	43:
		//Validate the CA group track length
		IF _XtsSystem.Environment.P_CaGroupOids[i] = _XtsSystem.AxesGroupRef.NcToPlc.CA.Common.GroupOID THEN
			IF _XtsSystem.Environment.Mc2CaGroup(UDINT_TO_UINT(i)).GetRailLength() <> _TrackCollection.Tracks.GetById(0).Length THEN
				LogSource.SourceName := 'InitializeXtsTask';
				LogMessage.Message	 := 'AxesGroupRef Length does not match Xts Track length!';
				LogMessage.MessageId := E_XtsLogMessage.SystemInitializationAxesGroupLengthMismatch;
				LogMessage.Severity	 := 3;
				_Logger.LogMessageInstance(LogSource, LogMessage);
				Trace.LogMessage(Key	   := LogSource.SourceName,
								 Value	   := LogMessage.Message,
								 MessageId := LogMessage.MessageId,
								 Severity  := LogMessage.Severity);

				_Error	 := TRUE;
				_ErrorId := E_XtsLogMessage.SystemInitializationAxesGroupLengthMismatch;
				_State	 := 65535;
			ELSE
				_State := 50;
			END_IF
		ELSE
			i := i + 1;
			IF i > _XtsSystem.Environment.P_CaGroupCount THEN
				LogSource.SourceName := 'InitializeXtsTask';
				LogMessage.Message	 := 'No CA group found!';
				LogMessage.MessageId := E_XtsLogMessage.SystemInitializationAxesGroupNotFound;
				LogMessage.Severity	 := 3;
				_Logger.LogMessageInstance(LogSource, LogMessage);
				Trace.LogMessage(Key	   := LogSource.SourceName,
								 Value	   := LogMessage.Message,
								 MessageId := LogMessage.MessageId,
								 Severity  := LogMessage.Severity);

				_Error	 := TRUE;
				_ErrorId := E_XtsLogMessage.SystemInitializationAxesGroupLengthMismatch;
				_State	 := 65535;
			END_IF
		END_IF

	50:
		_XtsUtility.Utility := _Xpu;
		_State				:= 60;

	60:
		IF PartSetup() THEN
			_XtsSystem.ManualDiagnoser.RefreshCollections := TRUE;
			_State										  := 100;
		END_IF

	100:
		LogSource.SourceName := 'InitializeXtsTask';
		LogMessage.Message	 := 'Initialization Finished.';
		LogMessage.MessageId := E_XtsLogMessage.SystemInitializationFinished;
		LogMessage.Severity	 := 1;
		_Logger.LogMessageInstance(LogSource, LogMessage);
		_Initialized	 := TRUE;
		_Busy			 := FALSE;
		_CommandExecuted := FALSE;
		_State			 := 0;
END_CASE
END_METHOD

{attribute 'monitoring':='call'}
PROPERTY Initialized : BOOL
GET
Initialized := _Initialized;
END_GET
SET
_Initialized := Initialized;
END_SET
END_PROPERTY

METHOD PRIVATE InfoServerSetup : BOOL
VAR_INPUT
END_VAR
CASE _SubState OF
	0:
		IF _XtsEnvironment.P_InfoServerCount > 0 THEN
			_InfoServer := _XtsEnvironment.InfoServerTcIo(1); //TODO: This needs to handle > 1 Infoserver
			_SubState		:= 10;
		ELSE
			InfoServerSetup := TRUE;
		END_IF
	10:
		IF _XtsEnvironment.GetInfoServerOids(TRUE) THEN
			_XtsEnvironment.GetInfoServerOids(FALSE);
			_InfoServerOTCID := _XtsEnvironment.P_InfoServerOids[1];
			_SubState := 20;
		END_IF
	20:
		IF _InfoServer.Init(TRUE,_InfoServerOTCID) THEN
			_InfoServer.Init(FALSE,_InfoServerOTCID);
			_SubState := 0;
			InfoServerSetup := TRUE;
		END_IF
END_CASE
END_METHOD

METHOD MoverSetup : BOOL
VAR
	LogSource  : TraceSourceInfo;
	LogMessage : TraceMessageInfo;
END_VAR
LogSource.SourceName := 'InitializeXtsTask';
LogMessage.Message	 := 'Mover Initialization Started.';
LogMessage.MessageId := E_XtsLogMessage.SystemMoverInitializationFinished;
LogMessage.Severity	 := 0;
_Logger.LogMessageInstance(LogSource, LogMessage);
_XtsSystem.Movers.ResetIterator();
WHILE _XtsSystem.Movers.MoveToNext DO
	IF _XtsSystem.Movers.Current.VirtualMover THEN
		CONTINUE;
	END_IF

	_XtsSystem.Movers.Current.MoverUtility := _Xpu.MoverTcIo(UDINT_TO_UINT(_XtsSystem.Movers.CurrentItem));
	_XtsSystem.Movers.Current.RefreshMoverId(_Xpu);
END_WHILE

_XtsUtilityProperties.UtilityProperties.Mover.XtsMoverType		 := _Xpu.GetMoverType();
_XtsUtilityProperties.UtilityProperties.Mover.XtsMagnetPlateType := _Xpu.GetMagnetPlateType();
MoverSetup														 := TRUE;
END_METHOD

METHOD PartSetup : BOOL
VAR_INPUT
END_VAR

VAR
	pPart	   : POINTER TO XtsPart;
	Part	   : I_XtsPart;
	_Parent	   : I_ContainModules;
	LogSource  : TraceSourceInfo;
	LogMessage : TraceMessageInfo;
END_VAR
CASE _SubState OF
	0:
		LogSource.SourceName := 'InitializeXtsTask';
		LogMessage.Message	 := 'Part Initialization Started.';
		LogMessage.MessageId := E_XtsLogMessage.SystemMoverInitializationStarted;
		LogMessage.Severity	 := 0;
		_Logger.LogMessageInstance(LogSource, LogMessage);
		IF NOT _Xpu.GetPartOids() THEN
			RETURN;
		END_IF

		IF _Xpu.P_PartCount < 1 THEN
			PartSetup := TRUE;
			RETURN;
		END_IF

		FOR i := 1 TO _Xpu.P_PartCount DO
			pPart		   := __NEW(XtsPart(Name := CONCAT('Part ', UDINT_TO_STRING(i))));
			Part		   := pPart^;
			Part.XtsPartId := UDINT_TO_UINT(i);
			Part.Utility   := _Xpu.PartTcIo(UDINT_TO_UINT(i));
			__QUERYINTERFACE(_XpuId, _Parent);
			Part.RegisterWithParent(_Parent);
			_PartCollection.Parts.AddItem(Part);
		END_FOR

		LogSource.SourceName := 'InitializeXtsTask';
		LogMessage.Message	 := CONCAT(TO_STRING(_PartCollection.Parts.Count), ' Parts Initialization Finished.');
		LogMessage.MessageId := E_XtsLogMessage.SystemPartInitializationFinished;
		LogMessage.Severity	 := 0;
		_Logger.LogMessageInstance(LogSource, LogMessage);
		PartSetup := TRUE;
		_SubState := 0;
END_CASE
END_METHOD

METHOD TrackSetup : BOOL
VAR_INPUT
END_VAR
VAR
	Track : I_XtsTrack;
	LogSource  : TraceSourceInfo;
	LogMessage : TraceMessageInfo;
	AxGroup : AXES_GROUP_REF;
END_VAR
CASE _SubState OF
	0:
		IF NOT _Xpu.GetTrackOids() THEN
			RETURN;
		END_IF

		IF NOT _TrackCollection.Tracks.IsEmpty THEN
			_TrackCollection.Tracks.Clear();
		END_IF

		LogSource.SourceName := 'InitializeXtsTask';
		LogMessage.Message	 := CONCAT(TO_STRING(_TrackCollection.Tracks.Count), ' Tracks Initialization Started.');
		LogMessage.MessageId := E_XtsLogMessage.SystemTrackInitializationStarted;
		_TrackCollection.Tracks.Create(_Xpu.P_TrackCount + 1);
		Track		   := _TrackCollection.Tracks.GetById(0);
		Track.Id	   := 0;
		Track.Length   := _Xpu.TrackTcIo(1).GetLength();
		Track.Otcid	   := 0;
		Track.Offset   := _Xpu.TrackTcIo(1).GetOffset();
		Track.Polarity := _Xpu.TrackTcIo(1).GetPolarity();
		Track.Utility  := 0;
		IF _Xpu.P_TrackCount = 0 THEN
			_SubState := 10;
			RETURN;
		END_IF

		FOR i := 1 TO _Xpu.P_TrackCount DO
			Track		   := _TrackCollection.Tracks.GetById(i);
			Track.Id	   := i;
			Track.Length   := _Xpu.TrackTcIo(UDINT_TO_UINT(i)).GetLength();
			Track.Otcid	   := _Xpu.P_TrackOids[i];
			Track.Offset   := _Xpu.TrackTcIo(UDINT_TO_UINT(i)).GetOffset();
			Track.Polarity := _Xpu.TrackTcIo(UDINT_TO_UINT(i)).GetPolarity();
			Track.Utility  := _Xpu.TrackTcIo(UDINT_TO_UINT(i));
		END_FOR

		_SubState := 10;

	10:
		_XtsSystem.Movers.ResetIterator();
		WHILE _XtsSystem.Movers.MoveToNext DO
			_XtsSystem.Movers.Current.Tracks := _TrackCollection.Tracks;
		END_WHILE

		LogSource.SourceName := 'InitializeXtsTask';
		LogMessage.Message	 := CONCAT(TO_STRING(_TrackCollection.Tracks.Count), ' Tracks Initialization Finished.');
		LogMessage.MessageId := E_XtsLogMessage.SystemTrackInitializationFinished;
		LogMessage.Severity	 := 0;
		_Logger.LogMessageInstance(LogSource, LogMessage);
		_SubState  := 0;
		TrackSetup := TRUE;
END_CASE
END_METHOD

//FB_Init is always available implicitly AND it is used primarily FOR initialization.

//The return value is not evaluated. For a specific influence, you can also declare the

//methods explicitly and provide additional code there with the standard initialization

//code. You can evaluate the return value.
METHOD FB_Init : BOOL
VAR_INPUT
	bInitRetains	: BOOL; // TRUE: the retain variables are initialized (reset warm / reset cold)
	bInCopyCode		: BOOL; // TRUE: the instance will be copied to the copy code afterward (online change)
END_VAR
_TaskName := 'Initalize Xts';
_TaskId	  := XtsSystemTaskId.INITIALIZE;
END_METHOD

METHOD Reset
_State			 := 0;
_Error			 := FALSE;
_ErrorId		 := 0;
_Busy			 := FALSE;
_CommandExecuted := FALSE;
_SubState		 := 0;
END_METHOD

{attribute 'monitoring' := 'call'}
PROPERTY XpuId : I_XtsXpuId
GET
XpuId := _XpuId;
END_GET
SET
_XpuId := XpuId;
__QUERYINTERFACE(_XpuId, _XtsSystem);
__QUERYINTERFACE(_XpuId, _PartCollection);
__QUERYINTERFACE(_XpuId, _TrackCollection);
__QUERYINTERFACE(_XpuId, _XtsUtilityProperties);
__QUERYINTERFACE(_XpuId, _XtsUtility);
__QUERYINTERFACE(_XtsSystem.TracePublisher,_Logger);
_MoverDetectTask   := _XtsSystem.XtsTasks.GetTaskById(XtsSystemTaskId.MOVER_DETECTION);
_MoverRedetectTask := _XtsSystem.XtsTasks.GetTaskById(XtsSystemTaskId.MOVER_REDETECTION);
_MoverIDTask	   := _XtsSystem.XtsTasks.GetTaskById(XtsSystemTaskId.MOVER_IDENTIFICATION);
END_SET
END_PROPERTY

END_FUNCTION_BLOCK

// _Internal/XtsSystem/Tasks/Interfaces/I_XtsInitializeTask
INTERFACE I_XtsInitializeTask EXTENDS I_XtsTask, I_Initializable, I_Resettable

END_INTERFACE

// _Internal/XtsSystem/Tasks/DisableXtsTask
{attribute 'no_explicit_call' := 'This FB is a CLASS and must be accessed using methods or properties'}
FUNCTION_BLOCK DisableXtsTask EXTENDS XtsTaskResult IMPLEMENTS I_XtsDisableTask, I_Cyclic
VAR
	_XpuId					   : I_XtsXpuId;
	_XtsSystem				   : I_XtsSystem;
	_State					   : UDINT;
	_MoverCommander			   : I_XtsMoverCommander;
	_GroupController		   : I_XtsMoverGroupController;
	_PositionTriggerCollection : I_XtsPositionTriggerCollection;
	_StationCollection		   : I_XtsStationCollection;
	_ZoneCollection			   : I_XtsZoneCollection;
	_AxesGroup				   : REFERENCE TO AXES_GROUP_REF;

	//CA Group Parameters
	_CollisionAvoidanceGroupParameters : I_CollisionAvoidanceGroupable;
END_VAR

PROPERTY AxesGroup : REFERENCE TO AXES_GROUP_REF
GET
AxesGroup REF= _AxesGroup;
END_GET
SET
_AxesGroup REF= AxesGroup;
END_SET
END_PROPERTY

METHOD CyclicLogic
VAR
	_Check	  : BOOL;
	AxesGroup : REFERENCE TO AXES_GROUP_REF;
	LogSource  : TraceSourceInfo;
	LogMessage : TraceMessageInfo;
END_VAR
CASE _State OF
	0:
		IF _CommandExecuted THEN
			_Busy	 := TRUE;
			_Error	 := FALSE;
			_ErrorId := 0;
			_GroupController.Disable();
			_State := 10;
		END_IF

	10:
		//Disable Group
		IF _GroupController.Error THEN
			_Error := TRUE;
			_State := 255;
		ELSIF NOT _GroupController.Enabled THEN
			AxesGroup REF= _AxesGroup;
			_MoverCommander.RemoveFromGroup(_XtsSystem.Movers, AxesGroup, 1);
			_State := 20;
		END_IF

	20:
		//Remove All From Group
		IF _MoverCommander.Error THEN
			_Error := TRUE;
			_State := 255;
		ELSIF NOT _MoverCommander.Busy THEN
			_MoverCommander.Disable(_XtsSystem.Movers);
			_State := 30;
		END_IF

	30:
		//Disable all movers
		IF _MoverCommander.Error THEN
			_Error := TRUE;
			_State := 255;
		ELSIF NOT _MoverCommander.Busy THEN
			_State := 40;
		END_IF

	40:
		//Disable All Stations
		IF NOT _XtsSystem.Config.CommandStationsOnDisable THEN
			LogSource.SourceName := 'DisableXtsTask';
			LogMessage.Message	 := 'Station Disable Skipped due to configuration.';
			LogMessage.MessageId := E_XtsLogMessage.SystemDisableStationSkipped;
			LogMessage.Severity	 := 0;
			_Logger.LogMessageInstance(LogSource, LogMessage);
			_State := 50;
			RETURN;
		END_IF

		_StationCollection.ResetIterator();
		_Check := TRUE;
		WHILE _StationCollection.MoveToNext DO
			_StationCollection.Current.Disable();
			_Check := _Check AND NOT _StationCollection.Current.Enabled;
		END_WHILE

		IF _Check THEN
			_State := 50;
		END_IF

	50:
		IF NOT _XtsSystem.Config.CommandPositionTriggersOnDisable THEN
			LogSource.SourceName := 'DisableXtsTask';
			LogMessage.Message	 := 'PositionTrigger Disable Skipped due to configuration.';
			LogMessage.MessageId := E_XtsLogMessage.SystemDisableStationSkipped;
			LogMessage.Severity	 := 0;
			_Logger.LogMessageInstance(LogSource, LogMessage);
			_State := 60;
			RETURN;
		END_IF

		//Disable All Position Triggers
		_PositionTriggerCollection.ResetIterator();
		_Check := TRUE;
		WHILE _PositionTriggerCollection.MoveToNext DO
			_PositionTriggerCollection.Current.Disable();
			_Check := _Check AND NOT _PositionTriggerCollection.Current.Enabled;
		END_WHILE

		IF _Check THEN
			_State := 60;
		END_IF

	60:
		_State			 := 0;
		_CommandExecuted := FALSE;
		_Busy			 := FALSE;
END_CASE
END_METHOD

METHOD Execute : I_XtsTaskResult
_CommandExecuted := TRUE;
Execute := THIS^;
END_METHOD

//FB_Init is always available implicitly and it is used primarily for initialization.

//The return value is not evaluated. For a specific influence, you can also declare the

//methods explicitly and provide additional code there with the standard initialization

//code. You can evaluate the return value.
METHOD FB_Init : BOOL
VAR_INPUT
	bInitRetains		  : BOOL; // TRUE: the retain variables are initialized (reset warm / reset cold)
	bInCopyCode			  : BOOL; // TRUE: the instance will be copied to the copy code afterward (online change)
END_VAR
_TaskName := 'Disable Xts';
_TaskId	  := XtsSystemTaskId.DISABLE;
END_METHOD

METHOD Reset
_State			 := 0;
_Error			 := FALSE;
_ErrorId		 := 0;
_Busy			 := FALSE;
_CommandExecuted := FALSE;
END_METHOD

{attribute 'monitoring' := 'call'}
PROPERTY XpuId : I_XtsXpuId
GET
XpuId := _XpuId;
END_GET
SET
_XpuId := XpuId;
__QUERYINTERFACE(_XpuId, _XtsSystem);
__QUERYINTERFACE(_XtsSystem.Parameters, _CollisionAvoidanceGroupParameters);
__QUERYINTERFACE(_XtsSystem.TracePublisher,_Logger);
_StationCollection		   := _XtsSystem.Stations;
_PositionTriggerCollection := _XtsSystem.PositionTriggers;
_ZoneCollection			   := _XtsSystem.Zones;
END_SET
END_PROPERTY

PROPERTY XtsMoverCommander : I_XtsMoverCommander
SET
_MoverCommander := XtsMoverCommander;
END_SET
END_PROPERTY

PROPERTY XtsMoverGroupController : I_XtsMoverGroupController
SET
_GroupController := XtsMoverGroupController;
END_SET
END_PROPERTY

END_FUNCTION_BLOCK

// _Internal/XtsSystem/Tasks/Interfaces/I_XtsDisableTask
INTERFACE I_XtsDisableTask EXTENDS I_XtsTask, I_ContainXtsMoverCommander, I_ContainXtsMoverGroupController, I_XtsExecutableTask, I_Resettable

PROPERTY AxesGroup : REFERENCE TO AXES_GROUP_REF
GET
END_GET
SET
END_SET
END_PROPERTY

END_INTERFACE

// _Internal/XtsSystem/Tasks/MoverDetectionTask
{attribute 'no_explicit_call' := 'This FB is a CLASS and must be accessed using methods or properties'}
FUNCTION_BLOCK MoverDetectionTask EXTENDS XtsTaskResult IMPLEMENTS I_XtsMoverDetectionTask
VAR
	_XpuId : I_XtsXpuId;
	_Xpu   : I_ContainXtsUtility;
END_VAR

METHOD Execute : I_XtsTaskResult
Execute := THIS^;
_Xpu.Utility.TriggerDetection();
END_METHOD

//FB_Init is always available implicitly and it is used primarily for initialization.

//The return value is not evaluated. For a specific influence, you can also declare the

//methods explicitly and provide additional code there with the standard initialization

//code. You can evaluate the return value.
METHOD FB_Init : BOOL
VAR_INPUT
	bInitRetains		  : BOOL; // TRUE: the retain variables are initialized (reset warm / reset cold)
	bInCopyCode			  : BOOL; // TRUE: the instance will be copied to the copy code afterward (online change)
END_VAR
_TaskName := 'Mover Detection';
_TaskId	  := XtsSystemTaskId.MOVER_DETECTION;
END_METHOD

{attribute 'monitoring' := 'call'}
PROPERTY XpuId : I_XtsXpuId
GET
XpuId := _XpuId;
END_GET
SET
VAR
	_XtsSystem	   : I_XtsSystem;
END_VAR
_XpuId := XpuId;
__QUERYINTERFACE(_XpuId, _XtsSystem);
__QUERYINTERFACE(_XtsSystem.TracePublisher, _Logger);
__QUERYINTERFACE(_XpuId, _Xpu);
END_SET
END_PROPERTY

END_FUNCTION_BLOCK

// _Internal/XtsSystem/Tasks/Interfaces/I_XtsMoverDetectionTask
INTERFACE I_XtsMoverDetectionTask EXTENDS I_XtsTask, I_XtsExecutableTask

END_INTERFACE

// _Internal/XtsSystem/Tasks/MoverRedetectionTask
{attribute 'no_explicit_call' := 'This FB is a CLASS and must be accessed using methods or properties'}
FUNCTION_BLOCK MoverRedetectionTask EXTENDS XtsTaskResult IMPLEMENTS I_XtsMoverRedetectionTask
VAR
	_XpuId : I_XtsXpuId;
	_Xpu   : I_ContainXtsUtility;
END_VAR

METHOD Execute : I_XtsTaskResult
Execute := THIS^;
_Xpu.Utility.TriggerRedetection();
END_METHOD

//FB_Init is always available implicitly and it is used primarily for initialization.

//The return value is not evaluated. For a specific influence, you can also declare the

//methods explicitly and provide additional code there with the standard initialization

//code. You can evaluate the return value.
METHOD FB_Init : BOOL
VAR_INPUT
	bInitRetains		  : BOOL; // TRUE: the retain variables are initialized (reset warm / reset cold)
	bInCopyCode			  : BOOL; // TRUE: the instance will be copied to the copy code afterward (online change)
END_VAR
_TaskName := 'Mover Redetection';
_TaskId	  := XtsSystemTaskId.MOVER_REDETECTION;
END_METHOD

{attribute 'monitoring' := 'call'}
PROPERTY XpuId : I_XtsXpuId
GET
XpuId := _XpuId;
END_GET
SET
VAR
	_XtsSystem : I_XtsSystem;
END_VAR
_XpuId := XpuId;
__QUERYINTERFACE(_XpuId, _XtsSystem);
__QUERYINTERFACE(_XtsSystem.TracePublisher, _Logger);
__QUERYINTERFACE(_XpuId, _Xpu);
END_SET
END_PROPERTY

END_FUNCTION_BLOCK

// _Internal/XtsSystem/Tasks/Interfaces/I_XtsMoverRedetectionTask
INTERFACE I_XtsMoverRedetectionTask EXTENDS I_XtsTask, I_XtsExecutableTask

END_INTERFACE

// _Internal/XtsSystem/Tasks/MoverIdentificationTask
{attribute 'no_explicit_call' := 'This FB is a CLASS and must be accessed using methods or properties'}
FUNCTION_BLOCK MoverIdentificationTask EXTENDS XtsTaskResult IMPLEMENTS I_XtsMoverIdentificationTask
VAR
	_XtsSystem : I_XtsSystem;
	_XpuId	   : I_XtsXpuId;
	_Xpu	   : I_ContainXtsUtility;
	_Movers	   : I_XtsMoverEnumerator;
END_VAR

METHOD CyclicLogic
VAR
	DetectionValid : BOOL;
END_VAR
IF _Xpu.Utility = 0 AND _XtsSystem.Initialized THEN
	//TODO: Create an event/alarm
	_Error := TRUE;
	RETURN;
END_IF

IF _Busy THEN
	_Error := _Xpu.Utility.GetHasMoverIdDetectionError();

	//TODO: Create an event/alarm
	DetectionValid := _Xpu.Utility.GetIsMoverIdDetectionValid();
	IF DetectionValid THEN
		_Movers.ResetIterator();
		WHILE _Movers.MoveToNext DO
			_Movers.Current.RefreshMoverId(_XtsSystem.Utility);
		END_WHILE
	END_IF

	_Busy := NOT (DetectionValid OR _Error);
END_IF
END_METHOD

METHOD Execute : I_XtsTaskResult
Execute := THIS^;
IF _Xpu.Utility = 0 THEN
	_Error := TRUE;

	//TODO: Trigger error/log message that Xpu Utility is 0
END_IF

//Protect against repeated calls
IF _Busy THEN
	RETURN;
END_IF

IF _Xpu.Utility.GetMoverIdDetectionMode() = MoverIdDetectionMode.Standard THEN
	_Busy := FALSE;
	_Movers.ResetIterator();
	WHILE _Movers.MoveToNext DO
		_Movers.Current.RefreshMoverId(_XtsSystem.Utility);
	END_WHILE

	RETURN;
END_IF

_Error	 := FALSE;
_ErrorId := 0;
_Busy	 := TRUE;
_Xpu.Utility.TriggerMoverIdDetection();
END_METHOD

//FB_Init is always available implicitly and it is used primarily for initialization.

//The return value is not evaluated. For a specific influence, you can also declare the

//methods explicitly and provide additional code there with the standard initialization

//code. You can evaluate the return value.
METHOD FB_Init : BOOL
VAR_INPUT
	bInitRetains		  : BOOL; // TRUE: the retain variables are initialized (reset warm / reset cold)
	bInCopyCode			  : BOOL; // TRUE: the instance will be copied to the copy code afterward (online change)
END_VAR
_TaskName := 'Mover 1 Detection';
_TaskId	  := XtsSystemTaskId.MOVER_IDENTIFICATION;
END_METHOD

{attribute 'monitoring' := 'call'}
PROPERTY XpuId : I_XtsXpuId
GET
XpuId := _XpuId;
END_GET
SET
_XpuId := XpuId;
__QUERYINTERFACE(_XpuId, _XtsSystem);
__QUERYINTERFACE(_XtsSystem.TracePublisher, _Logger);
__QUERYINTERFACE(_XtsSystem.Movers, _Movers);
__QUERYINTERFACE(_XpuId, _Xpu);
END_SET
END_PROPERTY

END_FUNCTION_BLOCK

// _Internal/XtsSystem/Properties/XtsSystemConfiguration
FUNCTION_BLOCK XtsSystemConfiguration IMPLEMENTS I_XtsSystemConfiguration
VAR
	_CommandStationsOnEnable		  : BOOL := TRUE;
	_CommandPositionTriggersOnEnable  : BOOL := TRUE;
	_CommandStationsOnDisable		  : BOOL := TRUE;
	_CommandPositionTriggersOnDisable : BOOL := TRUE;
END_VAR

{attribute 'monitoring' := 'call'}
PROPERTY CommandPositionTriggersOnDisable : BOOL
GET
CommandPositionTriggersOnDisable  := _CommandPositionTriggersOnDisable;
END_GET
SET
_CommandPositionTriggersOnDisable  := CommandPositionTriggersOnDisable;
END_SET
END_PROPERTY

{attribute 'monitoring' := 'call'}
PROPERTY CommandPositionTriggersOnEnable : BOOL
GET
CommandPositionTriggersOnEnable  := _CommandPositionTriggersOnEnable;
END_GET
SET
_CommandPositionTriggersOnEnable  := CommandPositionTriggersOnEnable;
END_SET
END_PROPERTY

{attribute 'monitoring' := 'call'}
PROPERTY CommandStationsOnDisable : BOOL
GET
CommandStationsOnDisable := _CommandStationsOnDisable;
END_GET
SET
_CommandStationsOnDisable := CommandStationsOnDisable;
END_SET
END_PROPERTY

{attribute 'monitoring' := 'call'}
PROPERTY CommandStationsOnEnable : BOOL
GET
CommandStationsOnEnable := _CommandStationsOnEnable;
END_GET
SET
_CommandStationsOnEnable := CommandStationsOnEnable;
END_SET
END_PROPERTY

END_FUNCTION_BLOCK

// _Internal/GroupController/XtsGroupController
FUNCTION_BLOCK XtsGroupController EXTENDS CyclicComponent IMPLEMENTS I_XtsMoverGroupController
VAR
	_AxesGroup	  : REFERENCE TO AXES_GROUP_REF;
	_Enabled	  : BOOL;
	_EnableGroup  : MC_GroupEnable;
	_DisableGroup : MC_GroupDisable;
	_ResetGroup	  : MC_GroupReset;
	_Status		  : MC_GroupReadStatus;
	_ErrorRead	  : MC_GroupReadError;
END_VAR

METHOD Disable
VAR_INPUT
END_VAR
_DisableGroup.Execute := TRUE;
END_METHOD

METHOD Enable
VAR_INPUT
END_VAR
_EnableGroup.Execute := TRUE;
END_METHOD

METHOD Reset
VAR_INPUT
END_VAR
_DisableGroup.Execute := FALSE;
_EnableGroup.Execute  := FALSE;
_ErrorRead.Enable	  := FALSE;
_ResetGroup.Execute	  := _Status.Error OR _Status.GroupErrorStop AND NOT _ResetGroup.Error;
END_METHOD

METHOD Accept
VAR_INPUT
	ComponentVisitor	: Core.I_ComponentVisitor;
END_VAR
ComponentVisitor.VisitComponent(THIS^);
END_METHOD

{attribute 'monitoring' := 'call'}
PROPERTY AxesGroup : REFERENCE TO AXES_GROUP_REF
GET
AxesGroup REF= _AxesGroup;
END_GET
SET
_AxesGroup REF= AxesGroup;
END_SET
END_PROPERTY

{attribute 'monitoring':='call'}
PROPERTY Busy : BOOL
GET
END_GET
END_PROPERTY

METHOD CyclicLogic
IF NOT __ISVALIDREF(_AxesGroup) THEN
	RETURN;
END_IF

_Status.Enable	  := TRUE;
_ErrorRead.Enable := _Status.Error OR _Status.GroupErrorStop AND NOT _ErrorRead.Error;
_EnableGroup(AxesGroup := _AxesGroup);
_DisableGroup(AxesGroup := _AxesGroup);
_ResetGroup(AxesGroup := _AxesGroup);
_Status(AxesGroup := _AxesGroup);
_ErrorRead(AxesGroup := _AxesGroup);
IF _ResetGroup.Done OR _ResetGroup.Error THEN
	_ResetGroup.Execute := FALSE;
END_IF

IF _DisableGroup.Done THEN
	_Enabled			  := FALSE;
	_DisableGroup.Execute := FALSE;
END_IF

IF _EnableGroup.Done THEN
	_Enabled			 := TRUE;
	_EnableGroup.Execute := FALSE;
END_IF
END_METHOD

METHOD DeregisterWithParent
VAR_INPUT
	Parent	: Core.I_ContainComponents;
END_VAR
Parent.DeregisterCyclic(THIS^);
Parent.DeregisterComponent(THIS^);
END_METHOD

{attribute 'monitoring':='call'}
PROPERTY Done : BOOL
GET
VAR
	_Done  : BOOL;
	Status : I_XtsMoverTaskResult;
END_VAR
END_GET
END_PROPERTY

{attribute 'monitoring' := 'call'}
PROPERTY Enabled : BOOL
GET
Enabled := _Enabled;
END_GET
END_PROPERTY

{attribute 'monitoring':='call'}
PROPERTY Error : BOOL
GET
Error := _Status.GroupErrorStop OR _ResetGroup.Error;
END_GET
END_PROPERTY

{attribute 'monitoring':='call'}
PROPERTY ErrorId : UDINT
GET
IF _ResetGroup.Error THEN
	ErrorId := _ResetGroup.ErrorId;
END_IF

IF _ErrorRead.Valid AND _ErrorRead.GroupErrorId <> 0 THEN
	ErrorId := _ErrorRead.GroupErrorId;
END_IF
END_GET
END_PROPERTY

{attribute 'monitoring':='call'}
PROPERTY GroupStatus : E_MoverGroupState
GET
GroupStatus := E_MoverGroupState.Disabled;
IF NOT _Status.Valid THEN
	RETURN;
END_IF

IF _Status.GroupDisabled THEN
	GroupStatus := E_MoverGroupState.Disabled;
ELSIF _Status.GroupNotReady THEN
	GroupStatus := E_MoverGroupState.NotReady;
ELSIF _Status.GroupStandby THEN
	GroupStatus := E_MoverGroupState.Standby;
ELSIF _Status.GroupMoving THEN
	GroupStatus := E_MoverGroupState.Moving;
ELSIF _Status.GroupStopping THEN
	GroupStatus := E_MoverGroupState.Stopping;
ELSIF _Status.GroupErrorStop THEN
	GroupStatus := E_MoverGroupState.Error;
END_IF
END_GET
END_PROPERTY

METHOD RegisterWithParent
VAR_INPUT
	Parent	: Core.I_ContainComponents;
END_VAR
Parent.RegisterCyclic(THIS^);
Parent.RegisterComponent(THIS^);
END_METHOD

{attribute 'monitoring' := 'call'}
PROPERTY TaskName : STRING
GET
TaskName := _Name;
END_GET
END_PROPERTY

END_FUNCTION_BLOCK

// _Internal/Collections/Parts/PartCollection/XtsPartCollection
{attribute 'no_explicit_call' := 'This FB is a CLASS and must be accessed using methods or properties'}
FUNCTION_BLOCK XtsPartCollection IMPLEMENTS I_XtsPartCollection, I_Peekable
VAR
	_Collection : Collection;
END_VAR

{attribute 'monitoring':='call'}
PROPERTY Current : I_XtsPart
GET
__QUERYINTERFACE(_Collection.Current,Current);
END_GET
END_PROPERTY

{attribute 'monitoring' := 'call'}
PROPERTY CurrentItem : UDINT
GET
CurrentItem := _Collection.CurrentItem;
END_GET
END_PROPERTY

PROPERTY MoveToNext : BOOL
GET
MoveToNext := _Collection.MoveToNext;
END_GET
END_PROPERTY

METHOD ResetIterator
_Collection.ResetIterator();
END_METHOD

METHOD AcceptPeeker
VAR_INPUT
	Peeker	: Core.I_Peeker;
END_VAR
Peeker.PeekCollection(_Collection);
END_METHOD

METHOD AddItem
VAR_INPUT
	Part : I_XtsPart;
END_VAR
_Collection.AddItem(Part);
END_METHOD

METHOD Clear
VAR_INPUT
END_VAR
_Collection.Clear();
END_METHOD

{attribute 'monitoring' := 'call'}
PROPERTY Count : UDINT
GET
Count := _Collection.Count;
END_GET
END_PROPERTY

//FB_Exit must be implemented explicitly. If there is an implementation, then the
//method is called before the controller removes the code of the function block instance
//(implicit call). The return value is not evaluated.
METHOD FB_Exit: BOOL
VAR_INPUT
    bInCopyCode: BOOL;  // TRUE: the exit method is called in order to leave the instance which will be copied afterwards (online change).  
END_VAR
IF bInCopyCode OR IsEmpty THEN
	RETURN;
END_IF

ResetIterator();
WHILE MoveToNext DO
	Current.Dispose();
END_WHILE
Clear();
END_METHOD

METHOD GetById : I_XtsPart
VAR_INPUT
	PartId : UDINT;
END_VAR
VAR
	_Part : I_XtsPart;
END_VAR
GetById := NullObjects.XtsPart;
_Collection.ResetIterator();
WHILE _Collection.MoveToNext DO
	__QUERYINTERFACE(_Collection.Current,_Part);
	IF _Part.XtsPartId = UDINT_TO_UINT(PartId) THEN
		GetById := _Part;
		RETURN;
	END_IF
END_WHILE
END_METHOD

METHOD GetByOtcid : I_XtsPart
VAR_INPUT
	PartOtcid : OTCID;
END_VAR
VAR
	_Part : I_XtsPart;
END_VAR
__QUERYINTERFACE(NullObjects.XtsPart, GetByOtcid);
_Collection.ResetIterator();
WHILE _Collection.MoveToNext DO
	__QUERYINTERFACE(_Collection.Current, _Part);
	IF _Part.Properties.General.OTCID = PartOtcid THEN
		GetByOtcid := _Part;
		RETURN;
	END_IF
END_WHILE
END_METHOD

{attribute 'monitoring':='call'}
PROPERTY IsEmpty : BOOL
GET
IsEmpty := _Collection.IsEmpty;
END_GET
END_PROPERTY

METHOD Remove
VAR_INPUT
	Part : I_XtsPart;
END_VAR
_Collection.RemoveItem(Part);
END_METHOD

END_FUNCTION_BLOCK

// _Internal/XtsSystem/Status/XtsSystemStatus
{attribute 'no_explicit_call' := 'This FB is a CLASS and must be accessed using methods or properties'}
FUNCTION_BLOCK XtsSystemStatus IMPLEMENTS I_XtsSystemStatus
VAR
	_XtsSystem			 : I_XtsSystem;
	_Vdc24Okay			 : BOOL;
	_Vdc48Okay			 : BOOL;
	_PartReadyCounter	 : USINT;
	_PartNotReadyCounter : USINT;
END_VAR

METHOD CyclicLogic
VAR
	Part : I_XtsPart;
END_VAR
//TODO: Split this into a seperate set of commands
_Vdc24Okay := _XtsSystem.Utility.GetIsDcLinkVoltageReady();
_Vdc48Okay := _XtsSystem.Utility.GetIsDcLinkVoltageReady();
END_METHOD

//FB_Init is always available implicitly and it is used primarily for initialization.

//The return value is not evaluated. For a specific influence, you can also declare the

//methods explicitly and provide additional code there with the standard initialization

//code. You can evaluate the return value.
METHOD FB_Init : BOOL
VAR_INPUT
	bInitRetains : BOOL; // TRUE: the retain variables are initialized (reset warm / reset cold)
	bInCopyCode	 : BOOL; // TRUE: the instance will be copied to the copy code afterward (online change)   
	XtsSystem	 : I_XtsSystem;
END_VAR
_XtsSystem := XtsSystem;
END_METHOD

{attribute 'monitoring' := 'call'}
PROPERTY NumberOfMovers : UDINT
GET
NumberOfMovers := _XtsSystem.Movers.Count;
END_GET
END_PROPERTY

{attribute 'monitoring' := 'call'}
PROPERTY NumberOfParts : UDINT
GET
NumberOfParts := _XtsSystem.Parts.Count;
END_GET
END_PROPERTY

{attribute 'monitoring' := 'call'}
PROPERTY NumberOfPositionTriggers : UDINT
GET
NumberOfPositionTriggers := _XtsSystem.PositionTriggers.Count;
END_GET
END_PROPERTY

{attribute 'monitoring' := 'call'}
PROPERTY NumberOfStations : UDINT
GET
NumberOfStations := _XtsSystem.Stations.Count;
END_GET
END_PROPERTY

{attribute 'monitoring' := 'call'}
PROPERTY NumberOfTracks : UDINT
GET
NumberOfTracks := _XtsSystem.Tracks.Count;
END_GET
END_PROPERTY

{attribute 'monitoring' := 'call'}
PROPERTY NumberOfZones : UDINT
GET
NumberOfZones := _XtsSystem.Zones.Count;
END_GET
END_PROPERTY

{attribute 'monitoring':='call'}
PROPERTY NumberPartsNotReady : USINT
GET
NumberPartsNotReady := _PartNotReadyCounter;
END_GET
END_PROPERTY

{attribute 'monitoring':='call'}
PROPERTY NumberPartsReady : USINT
GET
NumberPartsReady := _PartReadyCounter;
END_GET
END_PROPERTY

{attribute 'monitoring':='call'}
PROPERTY Simulated : BOOL
GET
IF _XtsSystem.Utility = 0 THEN
	RETURN;
END_IF

Simulated := _XtsSystem.Utility.GetOperationMode() = OperationMode.Simulation;
END_GET
END_PROPERTY

{attribute 'monitoring':='call'}
PROPERTY Vdc24Okay : BOOL
GET
VAR
	VoltageOk : BOOL;
END_VAR
Vdc24Okay := _Vdc24Okay;
END_GET
END_PROPERTY

{attribute 'monitoring':='call'}
PROPERTY Vdc48Okay : BOOL
GET
Vdc48Okay := _Vdc48Okay;
END_GET
END_PROPERTY

END_FUNCTION_BLOCK

// _Internal/Collections/Tracks/TrackCollection/XtsTrackCollection
{attribute 'no_explicit_call' := 'This FB is a CLASS and must be accessed using methods or properties'}
{attribute 'hide_all_locals}
FUNCTION_BLOCK XtsTrackCollection IMPLEMENTS I_XtsTrackCollection
VAR
	pTrackBuffer	: POINTER TO PVOID;
	_NumberOfTracks : UINT;
	_CurrentTrack : I_XtsTrack;
	_CurrentIndex : UDINT := 0;
END_VAR

METHOD Clear
VAR
	i	   : UDINT;
	Track : POINTER TO XtsTrack;
END_VAR
IF IsEmpty THEN
	RETURN;
END_IF

FOR i := 0 TO _NumberOfTracks - 1 DO
	Track := GetTrackInstance(i);
	Track^.Dispose();
END_FOR

__DELETE(pTrackBuffer);
_NumberOfTracks := 0;
END_METHOD

{attribute 'monitoring' := 'call'}
PROPERTY Count : UDINT
GET
Count := _NumberOfTracks;
END_GET
END_PROPERTY

{attribute 'hide'}
METHOD Create : BOOL
VAR_INPUT
	NumberOfTracks : UINT;
END_VAR
VAR
	i		 : UINT;
	pTrack	 : POINTER TO XtsTrack;
	ppBuffer : POINTER TO POINTER TO XtsTrack;
END_VAR
IF NOT IsEmpty THEN
	Clear();
END_IF

_NumberOfTracks := NumberOfTracks;
pTrackBuffer	:= __NEW(PVOID, _NumberOfTracks);
IF pTrackBuffer <> 0 THEN
	FOR i := 0 TO _NumberOfTracks - 1 DO
		pTrack	  := __NEW(XtsTrack);
		ppBuffer  := pTrackBuffer + (i * SIZEOF(PVOID));
		ppBuffer^ := pTrack;
	END_FOR

	Create := TRUE;
END_IF
END_METHOD

METHOD GetById : I_XtsTrack
VAR_INPUT
	TrackId : UDINT;
END_VAR
GetById := GetTrackInstance(TrackId)^;
END_METHOD

METHOD GetByOtcid : I_XtsTrack
VAR_INPUT
	TrackOtcid : OTCID;
END_VAR
VAR
	i : UDINT;
	ppTrack : POINTER TO POINTER TO XtsTrack;
END_VAR
GetByOtcid := NullObjects.XtsTrack;
FOR i := 0 TO _NumberOfTracks - 1 DO
	ppTrack := pTrackBuffer + ((i) * SIZEOF(PVOID));
	IF ppTrack^^.Otcid = TrackOtcid THEN
		GetByOtcid := ppTrack^^;
		RETURN;
	END_IF
END_FOR
END_METHOD

{attribute 'monitoring' := 'call'}
PROPERTY IsEmpty : BOOL
GET
IsEmpty := _NumberOfTracks = 0;
END_GET
END_PROPERTY

{attribute 'monitoring' := 'call'}
PROPERTY Current : I_XtsTrack
GET
IF  _CurrentTrack = 0 THEN
	Current := NullObjects.XtsTrack;
ELSE
	Current := _CurrentTrack;
END_IF
END_GET
END_PROPERTY

{attribute 'monitoring' := 'call'}
PROPERTY CurrentIndex : UDINT
GET
CurrentIndex := _CurrentIndex;
END_GET
END_PROPERTY

PROPERTY MoveToNext : BOOL
GET
MoveToNext := FALSE;
IF _NumberOfTracks = 0 THEN
	RETURN;
END_IF

IF _CurrentIndex = _NumberOfTracks THEN
	RETURN;
END_IF

_CurrentTrack := GetById(_CurrentIndex + 1);
_CurrentIndex := _CurrentIndex + 1;
MoveToNext	  := TRUE;
END_GET
END_PROPERTY

METHOD ResetIterator
_CurrentTrack := NullObjects.XtsTrack;
_CurrentIndex := 0;
END_METHOD

METHOD PROTECTED CheckTrackId : BOOL
VAR_INPUT
	TrackId : UDINT;
END_VAR
CheckTrackId := (TrackId >= 0) AND (TrackId < _NumberOfTracks) AND (pTrackBuffer <> 0);
END_METHOD

METHOD PROTECTED GetTrackInstance : POINTER TO XtsTrack
VAR_INPUT
	TrackId : UDINT;
END_VAR

VAR
	ppTrack : POINTER TO POINTER TO XtsTrack;
END_VAR
IF CheckTrackId(TrackId) THEN
	ppTrack := pTrackBuffer + ((TrackId) * SIZEOF(PVOID));
	GetTrackInstance := ppTrack^;
ELSE
	GetTrackInstance := ADR(NullObjects.XtsTrack);
END_IF
END_METHOD

//FB_Exit must be implemented explicitly. If there is an implementation, then the
//method is called before the controller removes the code of the function block instance
//(implicit call). The return value is not evaluated.
METHOD FB_Exit: BOOL
VAR_INPUT
    bInCopyCode: BOOL;  // TRUE: the exit method is called in order to leave the instance which will be copied afterwards (online change).  
END_VAR
IF bInCopyCode THEN
	RETURN;
END_IF

Clear();
END_METHOD

END_FUNCTION_BLOCK

// _Internal/XtsSystem/Properties/XtsSystemUtilityProperties
{attribute 'no_explicit_call' := 'This FB is a CLASS and must be accessed using methods or properties'}
FUNCTION_BLOCK XtsSystemUtilityProperties IMPLEMENTS I_XtsSystemUtilityProperties
VAR
	_Mover : XtsSystemUtilityPropertiesMover;
END_VAR

PROPERTY Mover : I_XtsSystemUtilityPropertiesMover
GET
Mover := _Mover;
END_GET
END_PROPERTY

END_FUNCTION_BLOCK

// _Internal/XtsSystem/Properties/XtsSystemUtilityPropertiesMover
{attribute 'no_explicit_call' := 'This FB is a CLASS and must be accessed using methods or properties'}
FUNCTION_BLOCK XtsSystemUtilityPropertiesMover IMPLEMENTS I_XtsSystemUtilityPropertiesMover
VAR
	_MagnetPlate : MagnetPlateType;
	_MoverType	 : MoverType;
END_VAR

PROPERTY XtsMagnetPlateType : MagnetPlateType
GET
XtsMagnetPlateType := _MagnetPlate;
END_GET
SET
_MagnetPlate := XtsMagnetPlateType;
END_SET
END_PROPERTY

PROPERTY XtsMoverType : MoverType
GET
XtsMoverType := _MoverType;
END_GET
SET
_MoverType := XtsMoverType;
END_SET
END_PROPERTY

END_FUNCTION_BLOCK

// _Internal/Collections/Movers/MoverList/Interfaces/I_XtsMoverList
INTERFACE I_XtsMoverList EXTENDS I_XtsMoverCollection

METHOD Contains : BOOL
VAR_INPUT
	Mover : I_XtsMover;
END_VAR
END_METHOD

METHOD GetAtIndex : I_XtsMover
VAR_INPUT
	Index : UDINT; //0 indexed
END_VAR
END_METHOD

METHOD InsertAtIndex
VAR_INPUT
	Mover : I_XtsMover;
	Index : UDINT;
END_VAR
END_METHOD

METHOD RemoveAtIndex
VAR_INPUT
	MoverIndex : UDINT;
END_VAR
END_METHOD

END_INTERFACE

// _Internal/Collections/Movers/MoverList/XtsMoverList
{attribute 'no_explicit_call' := 'This FB is a CLASS and must be accessed using methods or properties'}
FUNCTION_BLOCK XtsMoverList IMPLEMENTS I_XtsMoverList
VAR
	_List : List;
END_VAR

METHOD AcceptMoverVisitor
VAR_INPUT
	MoverVisitor : I_XtsMoverVisitor;
END_VAR
VAR
	Mover : I_XtsMover;
END_VAR
_List.ResetIterator();
WHILE _List.MoveToNext DO
	__QUERYINTERFACE(_List.Current, Mover);
	Mover.AcceptMoverVisitor(MoverVisitor);
END_WHILE
END_METHOD

METHOD AddItem
VAR_INPUT
	Mover	: I_XtsMover;
END_VAR
_List.AddItem(Mover);
END_METHOD

METHOD Clear
_List.Clear();
END_METHOD

{attribute 'monitoring' := 'call'}
PROPERTY Count : UDINT
GET
Count := _List.Count;
END_GET
END_PROPERTY

{attribute 'monitoring' := 'call'}
PROPERTY IsEmpty : BOOL
GET
IsEmpty := _List.IsEmpty;
END_GET
END_PROPERTY

METHOD Map
VAR_INPUT
	Validator : I_XtsMoverValidator;
	Visitor	  : I_XtsMoverVisitor;
END_VAR
VAR
	Mover : I_XtsMover;
END_VAR
_List.ResetIterator();
WHILE _List.MoveToNext DO
	__QUERYINTERFACE(_List.Current, Mover);
	IF Validator.Valid(Mover) THEN
		Visitor.VisitMover(Mover);
	END_IF
END_WHILE
END_METHOD

METHOD Remove
VAR_INPUT
	Mover	: I_XtsMover;
END_VAR
_List.RemoveItem(Mover);
END_METHOD

{attribute 'monitoring':='call'}
PROPERTY Current : I_XtsMover
GET
VAR
	Mover : I_XtsMover;
END_VAR
__QUERYINTERFACE(_List.Current,Mover);
Current := Mover;
END_GET
END_PROPERTY

{attribute 'monitoring' := 'call'}
PROPERTY CurrentItem : UDINT
GET
CurrentItem := _List.CurrentItem;
END_GET
END_PROPERTY

PROPERTY MoveToNext : BOOL
GET
MoveToNext := _List.MoveToNext;
END_GET
END_PROPERTY

METHOD ResetIterator
_List.ResetIterator();
END_METHOD

METHOD Contains : BOOL
VAR_INPUT
	Mover	: I_XtsMover;
END_VAR
IF _List.Count = 0 THEN
	Contains := FALSE;
	RETURN;
END_IF
Contains := _List.ContainsItem(Mover);
END_METHOD

//FB_Exit must be implemented explicitly. If there is an implementation, then the
//method is called before the controller removes the code of the function block instance
//(implicit call). The return value is not evaluated.
METHOD FB_Exit: BOOL
VAR_INPUT
    bInCopyCode: BOOL;  // TRUE: the exit method is called in order to leave the instance which will be copied afterwards (online change).  
END_VAR
_List.FB_Exit(bInCopyCode);
END_METHOD

METHOD GetAtIndex : I_XtsMover
VAR_INPUT
	Index : UDINT; //0 based
END_VAR
__QUERYINTERFACE(_List.GetAtIndex(Index), GetAtIndex);
END_METHOD

METHOD InsertAtIndex
VAR_INPUT
	Mover : I_XtsMover;
	Index : UDINT;
END_VAR
_List.InsertAtIndex(Mover, Index);
END_METHOD

{attribute 'monitoring':='call'}
PROPERTY Movers : I_XtsMoverCollection
GET
Movers := THIS^;
END_GET
END_PROPERTY

METHOD RemoveAtIndex
VAR_INPUT
	MoverIndex	: UDINT;
END_VAR
_List.RemoveAtIndex(MoverIndex);
END_METHOD

END_FUNCTION_BLOCK

// _Internal/Collections/Movers/MoverQueue/XtsMoverQueue
{attribute 'no_explicit_call' := 'This FB is a CLASS and must be accessed using methods or properties'}
FUNCTION_BLOCK XtsMoverQueue IMPLEMENTS I_XtsMoverQueue
VAR
	_Queue			 : XtsMoverList;
END_VAR

{attribute 'monitoring':='call'}
PROPERTY Current : I_XtsMover
GET
Current := _Queue.Current;
END_GET
END_PROPERTY

{attribute 'monitoring' := 'call'}
PROPERTY CurrentItem : UDINT
GET
CurrentItem := _Queue.CurrentItem;
END_GET
END_PROPERTY

METHOD Map
VAR_INPUT
	Validator : I_XtsMoverValidator;
	Visitor	  : I_XtsMoverVisitor;
END_VAR
VAR
	Mover : I_XtsMover;
END_VAR
_Queue.ResetIterator();
WHILE _Queue.MoveToNext DO
	__QUERYINTERFACE(_Queue.Current, Mover);
	IF Validator.Valid(Mover) THEN
		Visitor.VisitMover(Mover);
	END_IF
END_WHILE
END_METHOD

PROPERTY MoveToNext : BOOL
GET
MoveToNext := _Queue.MoveToNext;
END_GET
END_PROPERTY

METHOD ResetIterator
_Queue.ResetIterator();
END_METHOD

METHOD AcceptMoverVisitor
VAR_INPUT
	MoverVisitor : I_XtsMoverVisitor;
END_VAR
VAR
	Mover : I_XtsMover;
END_VAR
_Queue.ResetIterator();
WHILE _Queue.MoveToNext DO
	__QUERYINTERFACE(_Queue.Current, Mover);
	Mover.AcceptMoverVisitor(MoverVisitor);
END_WHILE
END_METHOD

METHOD Clear
_Queue.Clear();
END_METHOD

{attribute 'monitoring':='call'}
PROPERTY Count : UDINT
GET
Count := _Queue.Count;
END_GET
END_PROPERTY

METHOD Dequeue : I_XtsMover
IF Count = 0 THEN
	RETURN;
END_IF
__QUERYINTERFACE(_Queue.GetAtIndex(0),Dequeue);
_Queue.RemoveAtIndex(0);
END_METHOD

METHOD Enqueue
VAR_INPUT
	Mover	: I_XtsMover;
END_VAR
_Queue.AddItem(Mover);
END_METHOD

//FB_Exit must be implemented explicitly. If there is an implementation, then the
//method is called before the controller removes the code of the function block instance
//(implicit call). The return value is not evaluated.
METHOD FB_Exit: BOOL
VAR_INPUT
    bInCopyCode: BOOL;  // TRUE: the exit method is called in order to leave the instance which will be copied afterwards (online change).  
END_VAR
_Queue.FB_Exit(bInCopyCode);
END_METHOD

{attribute 'monitoring':='call'}
PROPERTY Movers : I_XtsMoverCollection
GET
Movers := _Queue;
END_GET
END_PROPERTY

METHOD Peek : I_XtsMover
IF Count = 0 THEN
	RETURN;
END_IF
__QUERYINTERFACE(_Queue.GetAtIndex(0),Peek);
END_METHOD

END_FUNCTION_BLOCK

// _Internal/Collections/Movers/MoverQueue/XtsMoverUniqueQueue
{attribute 'no_explicit_call' := 'This FB is a CLASS and must be accessed using methods or properties'}
FUNCTION_BLOCK XtsMoverUniqueQueue EXTENDS XtsMoverQueue
VAR
END_VAR

METHOD Enqueue
VAR_INPUT
	Mover	: I_XtsMover;
END_VAR
IF _Queue.Contains(Mover) THEN
	RETURN;
END_IF
_Queue.AddItem(Mover);
END_METHOD

END_FUNCTION_BLOCK

// _Internal/Collections/I_ContainXtsMoverList
INTERFACE I_ContainXtsMoverList EXTENDS I_Base

{attribute 'monitoring':='call'}
PROPERTY Movers : I_XtsMoverList
GET
END_GET
END_PROPERTY

END_INTERFACE

// _Internal/Collections/I_OperatesOnMovers
INTERFACE I_OperatesOnMovers EXTENDS I_Base

PROPERTY Movers : I_XtsMoverCollection
SET
END_SET
END_PROPERTY

END_INTERFACE

// _Internal/Frames/Interfaces/I_BaseFrame
INTERFACE I_BaseFrame EXTENDS I_Base

{attribute 'monitoring':='call'}
PROPERTY FrameName : STRING
GET
END_GET
SET
END_SET
END_PROPERTY

END_INTERFACE

// _Internal/Frames/Interfaces/I_FrameModulo
INTERFACE I_FrameModulo EXTENDS I_Base

{attribute 'monitoring' := 'call'}
PROPERTY ModuloLength : LREAL
GET
END_GET
SET
END_SET
END_PROPERTY

END_INTERFACE

// _Internal/Frames/Interfaces/I_FrameOffset
INTERFACE I_FrameOffset EXTENDS I_Base

{attribute 'monitoring' := 'call'}
PROPERTY OffsetToParent : LREAL
GET
END_GET
SET
END_SET
END_PROPERTY

END_INTERFACE

// _Internal/Frames/Interfaces/I_HasAReferenceFrame
INTERFACE I_HasAReferenceFrame EXTENDS I_Base

{attribute 'monitoring' := 'call'}
PROPERTY ReferenceFrame : I_ReferenceFrame
GET
END_GET
END_PROPERTY

METHOD SetReferenceFrame
VAR_INPUT
	ReferenceFrame : I_ReferenceFrame;
END_VAR
END_METHOD

END_INTERFACE

// _Internal/Frames/ReferenceFrame
{attribute 'no_explicit_call' := 'This FB is a CLASS and must be accessed using methods or properties'}
FUNCTION_BLOCK ReferenceFrame IMPLEMENTS I_ReferenceFrame
VAR
	{attribute 'hide'}
	NullReferenceFrame : NullReferenceFrame;
	_FrameName		   : T_MaxString;
	_OffsetToParent	   : LREAL;
	_ModuloLength	   : LREAL;
	_ReferenceFrame	   : I_ReferenceFrame := NullReferenceFrame;
END_VAR

//FB_Init is always available implicitly and it is used primarily for initialization.

//The return value is not evaluated. For a specific influence, you can also declare the

//methods explicitly and provide additional code there with the standard initialization

//code. You can evaluate the return value.
METHOD FB_Init : BOOL
VAR_INPUT
	bInitRetains   : BOOL; // TRUE: the retain variables are initialized (reset warm / reset cold)
	bInCopyCode	   : BOOL; // TRUE: the instance will be copied to the copy code afterward (online change)
	FrameName		   : T_MaxString;
	Offset		   : LREAL;
	ModuloLength   : LREAL;
	ReferenceFrame : I_ReferenceFrame;
END_VAR
_FrameName	  := FrameName;
_OffsetToParent		  := Offset;
_ModuloLength := ModuloLength;
IF ReferenceFrame <> 0 THEN
	_ReferenceFrame := ReferenceFrame;
END_IF
END_METHOD

{attribute 'monitoring' := 'call'}
PROPERTY FrameName : STRING
GET
FrameName := _FrameName;
END_GET
SET
FrameName := _FrameName;
END_SET
END_PROPERTY

{attribute 'monitoring' := 'call'}
PROPERTY ModuloLength : LREAL
GET
ModuloLength := _ModuloLength;
END_GET
SET
_ModuloLength := ModuloLength;
END_SET
END_PROPERTY

{attribute 'hide'}
PROPERTY OffsetToGlobal : LREAL
GET
OffsetToGlobal := _OffsetToParent + _ReferenceFrame.OffsetToGlobal;
END_GET
END_PROPERTY

{attribute 'monitoring' := 'call'}
PROPERTY OffsetToParent : LREAL
GET
OffsetToParent := _OffsetToParent;
END_GET
SET
_OffsetToParent := OffsetToParent;
END_SET
END_PROPERTY

{attribute 'monitoring' := 'call'}
PROPERTY ReferenceFrame : I_ReferenceFrame
GET
ReferenceFrame := _ReferenceFrame;
END_GET
END_PROPERTY

METHOD SetReferenceFrame 
VAR_INPUT
	ReferenceFrame	: I_ReferenceFrame;
END_VAR
_ReferenceFrame := ReferenceFrame;
END_METHOD

END_FUNCTION_BLOCK

// _Internal/Frames/Interfaces/I_ReferenceFrame
INTERFACE I_ReferenceFrame EXTENDS I_BaseFrame,I_FrameModulo,I_FrameOffset, I_HasAReferenceFrame, I_InGlobalSpace

END_INTERFACE

// _Internal/Frames/Interfaces/I_InGlobalSpace
INTERFACE I_InGlobalSpace EXTENDS I_Base

{attribute 'hide'}
PROPERTY OffsetToGlobal : LREAL
GET
END_GET
END_PROPERTY

END_INTERFACE

// _Internal/NullObjects/NullReferenceFrame
{attribute 'no_explicit_call' := 'This FB is a CLASS and must be accessed using methods or properties'}
{attribute 'conditionalshow'}
{warning disable C0094}
{warning disable C0568}
FUNCTION_BLOCK NullReferenceFrame IMPLEMENTS I_ReferenceFrame, I_NullObject
VAR
END_VAR

{attribute 'monitoring' := 'call'}
PROPERTY FrameName : STRING
GET
FrameName := 'Null Frame';
END_GET
SET
END_SET
END_PROPERTY

PROPERTY ModuloLength : LREAL
GET
END_GET
SET
END_SET
END_PROPERTY

PROPERTY OffsetToGlobal : LREAL
GET
END_GET
END_PROPERTY

PROPERTY OffsetToParent : LREAL
GET
END_GET
SET
END_SET
END_PROPERTY

PROPERTY ReferenceFrame : I_ReferenceFrame
GET
END_GET
END_PROPERTY

METHOD SetReferenceFrame
VAR_INPUT
	ReferenceFrame	: I_ReferenceFrame;
END_VAR
END_METHOD

END_FUNCTION_BLOCK

// _Internal/Frames/Interfaces/I_ReferencedPosition
INTERFACE I_ReferencedPosition EXTENDS I_Base, I_Positionable,I_HasAReferenceFrame

END_INTERFACE

// _Internal/Frames/ReferencedPosition
{attribute 'no_explicit_call' := 'This FB is a CLASS and must be accessed using methods or properties'}
FUNCTION_BLOCK ReferencedPosition IMPLEMENTS I_ReferencedPosition
VAR
	{attribute 'hide'}
	NullReferenceFrame : NullReferenceFrame;
	_GlobalPosition	   : LREAL;
	_CurrentFrame	   : I_ReferenceFrame := NullReferenceFrame;
	
	//
	_CurrentPosition   : LREAL;
END_VAR

{attribute 'monitoring' := 'call'}
PROPERTY Position : LREAL
GET
VAR
	tmp : LREAL;
END_VAR
tmp := _GlobalPosition - _CurrentFrame.OffsetToGlobal;
//If my current frame is modulo'd, return the position in that modulo
IF _CurrentFrame.ModuloLength <> 0.0 THEN
    tmp := tmp - _CurrentFrame.ModuloLength * TRUNC(tmp / _CurrentFrame.ModuloLength);
    IF tmp < 0.0 THEN
        tmp := tmp + _CurrentFrame.ModuloLength;
    END_IF; 
END_IF;
Position := tmp;
END_GET
SET
_GlobalPosition := Position + _CurrentFrame.OffsetToGlobal;
END_SET
END_PROPERTY

{attribute 'monitoring' := 'call'}
PROPERTY ReferenceFrame : I_ReferenceFrame
GET
END_GET
END_PROPERTY

METHOD SetReferenceFrame 
VAR_INPUT
	ReferenceFrame	: I_ReferenceFrame;
END_VAR
_CurrentFrame := ReferenceFrame;
END_METHOD

END_FUNCTION_BLOCK

// _Internal/NullObjects/NullAxisRef
{attribute 'no_explicit_call' := 'This FB is a CLASS and must be accessed using methods or properties'}
{attribute 'conditionalshow'}
{warning disable C0094}
FUNCTION_BLOCK NullAxisRef IMPLEMENTS I_AxisRef,I_NullObject
VAR
	NullAxis : AXIS_REF;
END_VAR

PROPERTY Axis : REFERENCE TO Tc2_MC2.AXIS_REF
GET
Axis REF= NullAxis;
END_GET
END_PROPERTY

END_FUNCTION_BLOCK

// _Internal/NullObjects/NullMechatronicsLocalLog
{attribute 'no_explicit_call' := 'This FB is a CLASS and must be accessed using methods or properties'}
{attribute 'conditionalshow'}
{warning disable C0094}
FUNCTION_BLOCK NullMechatronicsLocalLog IMPLEMENTS I_XtsLocalLog, I_NullObject
VAR
END_VAR

METHOD Clear
VAR_INPUT
END_VAR
END_METHOD

{attribute 'monitoring':='call'}
PROPERTY Commands : REFERENCE TO ARRAY[0..XtsCoreParameters.MAX_NUMBER_LOCAL_LOG - 1] OF T_MaxString
GET
END_GET
END_PROPERTY

{attribute 'monitoring':='call'}
PROPERTY DetailedCommands : REFERENCE TO ARRAY[0..XtsCoreParameters.MAX_NUMBER_LOCAL_LOG - 1] OF I_XtsLogCommand
GET
END_GET
END_PROPERTY

END_FUNCTION_BLOCK

// _Internal/NullObjects/NullMechatronicsLogger
{attribute 'no_explicit_call' := 'This FB is a CLASS and must be accessed using methods or properties'}
{attribute 'conditionalshow'}
{warning disable C0094}
FUNCTION_BLOCK NullMechatronicsLogger IMPLEMENTS I_XtsLogger, I_NullObject
VAR
END_VAR

METHOD LogMessage
VAR_INPUT
	Key	: Core.T_MaxString;
	Value	: Core.T_MaxString;
	SourceId	: UDINT := 0;
	TimeStamp	: ULINT := 0;
	MessageId	: UDINT := 1;
	Severity	: USINT := 1;
END_VAR
END_METHOD

METHOD LogMessageInstance
VAR_INPUT
	SourceInfo	: Core.I_TraceSourceInfo;
	MessageInfo	: Core.I_TraceMessageInfo;
	Arguments	: Core.I_TraceArgument := 0;
END_VAR
END_METHOD

END_FUNCTION_BLOCK

// _Internal/NullObjects/NullMechatronicsTracePublisher
{attribute 'no_explicit_call' := 'This FB is a CLASS and must be accessed using methods or properties'}
{attribute 'conditionalshow'}
{warning disable C0094}
FUNCTION_BLOCK NullMechatronicsTracePublisher IMPLEMENTS I_XtsTracePublisher, I_NullObject
VAR
END_VAR

METHOD LogMessage
VAR_INPUT
	Key	: Core.T_MaxString;
	Value	: Core.T_MaxString;
	SourceId	: UDINT := 0;
	TimeStamp	: ULINT := 0;
	MessageId	: UDINT := 1;
	Severity	: USINT := 1;
END_VAR
END_METHOD

METHOD LogMessageInstance
VAR_INPUT
	SourceInfo	: Core.I_TraceSourceInfo;
	MessageInfo	: Core.I_TraceMessageInfo;
	Arguments	: Core.I_TraceArgument := 0;
END_VAR
END_METHOD

METHOD Subscribe
VAR_INPUT
	Logger : I_XtsLogger;
END_VAR
END_METHOD

METHOD Unsubscribe
VAR_INPUT
	Logger : I_XtsLogger;
END_VAR
END_METHOD

END_FUNCTION_BLOCK

// _Internal/NullObjects/NullMoverCollection
{attribute 'no_explicit_call' := 'This FB is a CLASS and must be accessed using methods or properties'}
{attribute 'conditionalshow'}
{warning disable C0094}
{warning disable C0568}
FUNCTION_BLOCK NullMoverCollection IMPLEMENTS I_XtsMoverCollection, I_NullObject
VAR
END_VAR

METHOD AcceptMoverVisitor
VAR_INPUT
	MoverVisitor : I_XtsMoverVisitor;
END_VAR
END_METHOD

METHOD AddItem
VAR_INPUT
	Mover	: I_XtsMover;
END_VAR
END_METHOD

METHOD Clear
END_METHOD

PROPERTY Count : UDINT
GET
END_GET
END_PROPERTY

{attribute 'monitoring' := 'call'}
PROPERTY Current : I_XtsMover
GET
Current := NullObjects.XtsMover;
END_GET
END_PROPERTY

PROPERTY CurrentItem : UDINT
GET
END_GET
END_PROPERTY

{attribute 'monitoring' := 'call'}
PROPERTY IsEmpty : BOOL
GET
END_GET
END_PROPERTY

METHOD Map
VAR_INPUT
	Validator : I_XtsMoverValidator;
	Visitor	  : I_XtsMoverVisitor;
END_VAR
END_METHOD

PROPERTY MoveToNext : BOOL
GET
END_GET
END_PROPERTY

METHOD Remove
VAR_INPUT
	Mover	: I_XtsMover;
END_VAR
END_METHOD

METHOD ResetIterator
END_METHOD

END_FUNCTION_BLOCK

// _Internal/NullObjects/NullPositionTriggerCollection
{attribute 'no_explicit_call' := 'This FB is a CLASS and must be accessed using methods or properties'}
{attribute 'conditionalshow'}
{warning disable C0094}
{warning disable C0568}
FUNCTION_BLOCK NullPositionTriggerCollection IMPLEMENTS I_XtsPositionTriggerCollection, I_NullObject
VAR
END_VAR

METHOD AcceptXtsPositionTriggerVisitor
VAR_INPUT
	PositionTriggerVisitor : I_VisitXtsPositionTrigger;
END_VAR
END_METHOD

METHOD AddItem
VAR_INPUT
	PositionTrigger	: I_XtsPositionTrigger;
END_VAR
END_METHOD

METHOD Clear
END_METHOD

PROPERTY Count : UDINT
GET
END_GET
END_PROPERTY

{attribute 'monitoring' := 'call'}
PROPERTY Current : I_XtsPositionTrigger
GET
Current := NullObjects.XtsPositionTrigger;
END_GET
END_PROPERTY

PROPERTY CurrentItem : UDINT
GET
END_GET
END_PROPERTY

PROPERTY IsEmpty : BOOL
GET
END_GET
END_PROPERTY

PROPERTY MoveToNext : BOOL
GET
END_GET
END_PROPERTY

METHOD Remove
VAR_INPUT
	PositionTrigger	: I_XtsPositionTrigger;
END_VAR
END_METHOD

METHOD ResetIterator
END_METHOD

END_FUNCTION_BLOCK

// XtsPositionTrigger/XtsPositionTrigger
{attribute 'no_explicit_call' := 'This FB is a CLASS and must be accessed using methods or properties'}
FUNCTION_BLOCK XtsPositionTrigger EXTENDS CyclicComponent IMPLEMENTS I_XtsPositionTrigger
VAR
	{attribute 'hide'}
	_Enabled : BOOL;
	{attribute 'hide'}
	_RegisteredMovers		   : I_XtsMoverCollection;
	_DefaultMoverQueueBehavior : XtsMoverUniqueQueue;
	_MoverQueue				   : I_XtsMoverQueue := _DefaultMoverQueueBehavior;
	_DefaultPositionBehavior   : ReferencedPosition;
	_Position				   : I_Positionable := _DefaultPositionBehavior;
	{attribute 'hide'}
	_Status : XtsPositionTriggerStatus(THIS^, _DefaultMoverMonitorBehavior);

	//
	_DefaultMoverMonitorBehavior : MoverThresholdMonitorTask(THIS^);
	_MoverMonitor				 : I_MoverMonitor := _DefaultMoverMonitorBehavior;
	{attribute 'hide'}
	_LocalLogger : XtsLocalLogger;
	{attribute 'hide'}
	_Logger : XtsTracePublisher;
	{attribute 'hide'}
	LogMessage : TraceMessageInfo;
	{attribute 'hide'}
	LogSource : TraceSourceInfo;
END_VAR

//FB_Init is always available implicitly and it is used primarily for initialization.

//The return value is not evaluated. For a specific influence, you can also declare the

//methods explicitly and provide additional code there with the standard initialization

//code. You can evaluate the return value.
METHOD FB_Init : BOOL
VAR_INPUT
	bInitRetains	 : BOOL;						 // TRUE: the retain variables are initialized (reset warm / reset cold)
	bInCopyCode		 : BOOL;						 // TRUE: the instance will be copied to the copy code afterward (online change)
	Name			 : T_MaxString;					 //Name of the Station                       
	Position		 : LREAL := 0;					 //Position in mm the Station will be located
	RegisteredMovers : I_XtsMoverCollection;			 //Collection of Movers to Monitor
	System			 : I_ContainXtsPositionTriggers; //XtsSystem To Selfregister to
END_VAR
_Position.Position			  := Position;
_RegisteredMovers			  := RegisteredMovers;
_MoverMonitor.MonitoredMovers := _RegisteredMovers;
_Status.SetRegisteredMovers(RegisteredMovers);
IF System <> 0 THEN
	System.PositionTriggers.AddItem(THIS^);
	RegisterWithParent(System);
END_IF

LogSource.SourceName := Name;
_Logger.Subscribe(_LocalLogger);
IF XtsCoreParameters.TcEventLoggerEnabled THEN
	_Logger.Subscribe(XtsTrace.EventLogger);
END_IF
END_METHOD

METHOD Disable
VAR
	LogSource  : TraceSourceInfo;
	LogMessage : TraceMessageInfo;
END_VAR
_Enabled := FALSE;
LogSource.SourceName := _Name;
LogMessage.Message	 := 'Disabled.';
LogMessage.MessageId := E_XtsLogMessage.PositionTriggerDisabled;
_Logger.LogMessageInstance(LogSource, LogMessage);
END_METHOD

METHOD Enable
VAR
	LogSource  : TraceSourceInfo;
	LogMessage : TraceMessageInfo;
END_VAR
_Enabled := TRUE;
LogSource.SourceName := _Name;
LogMessage.Message	 := 'Enabled.';
LogMessage.MessageId := E_XtsLogMessage.PositionTriggerEnabled;
_Logger.LogMessageInstance(LogSource, LogMessage);
END_METHOD

{attribute 'monitoring' := 'call'}
PROPERTY Enabled : BOOL
GET
Enabled := _Enabled;
END_GET
END_PROPERTY

{attribute 'monitoring':='call'}
PROPERTY CommandLog : I_XtsLocalLog
GET
CommandLog := _LocalLogger;
END_GET
END_PROPERTY

PROPERTY TracePublisher : I_XtsTracePublisher
GET
TracePublisher := _Logger;
END_GET
END_PROPERTY

METHOD AcceptXtsPositionTriggerVisitor
VAR_INPUT
	PositionTriggerVisitor : I_VisitXtsPositionTrigger;
END_VAR
PositionTriggerVisitor.VisitXtsPositionTrigger(THIS^);
END_METHOD

METHOD CyclicLogic
VAR
	Mover : I_XtsMover;
END_VAR
IF NOT Enabled THEN
	RETURN;
END_IF
_MoverMonitor.CyclicLogic();
END_METHOD

//Deregisters Mover to be Monitored by Position Trigger
METHOD DeregisterMover
VAR_INPUT
	Mover : I_XtsMover; //Mover to Deregister
END_VAR
_RegisteredMovers.Remove(Mover);
LogSource.SourceName := _Name;
LogMessage.Message	 := CONCAT('Mover Deregistered: ', Mover.Name);
LogMessage.Severity	 := 0;
LogMessage.MessageId := E_XtsLogMessage.PositionTriggerMoverDeregistered;
_Logger.LogMessageInstance(LogSource, LogMessage);
END_METHOD

//Gets and Removes the First Mover in the Trigger Queue
METHOD GetMover : I_XtsMover
VAR
	LogMessage : TraceMessageInfo;
	LogSource  : TraceSourceInfo;
END_VAR
GetMover := _MoverMonitor.GetMover();
LogSource.SourceName := _Name;
LogMessage.Message	 := CONCAT('Get Mover called: ', GetMover.Name);
LogMessage.Severity	 := 10;
LogMessage.MessageId := E_XtsLogMessage.PositionTriggerGetMoverCalled;
_Logger.LogMessageInstance(LogSource, LogMessage);
END_METHOD

//Checks if provided Mover is currently registered and monitored
METHOD IsMoverRegistered : BOOL
VAR_INPUT
	Mover : I_XtsMover; //Mover to check
END_VAR
_RegisteredMovers.ResetIterator();
WHILE _RegisteredMovers.MoveToNext DO
	IF _RegisteredMovers.Current = Mover THEN
		IsMoverRegistered := TRUE;
		RETURN;
	END_IF
END_WHILE
END_METHOD

{attribute 'monitoring' := 'call'}
//True if a mover has crossed the Position Trigger
PROPERTY MoverIsPresent : BOOL
GET
MoverIsPresent := _MoverMonitor.MoverPresent;
END_GET
END_PROPERTY

{attribute 'monitoring' := 'call'}
//Queue of Movers that has crossed the Position Trigger
PROPERTY MoverQueue : I_XtsMoverQueue
GET
MoverQueue := _MoverQueue;
END_GET
END_PROPERTY

//Currently registered and monitored Movers
PROPERTY Movers : I_XtsMoverEnumerator
GET
Movers := _RegisteredMovers;
END_GET
SET
__QUERYINTERFACE(Movers,_RegisteredMovers); //upcasting
_MoverMonitor.MonitoredMovers := _RegisteredMovers;
_Status.SetRegisteredMovers(_RegisteredMovers);
END_SET
END_PROPERTY

{attribute 'monitoring' := 'call'}
//Location of the Position Trigger in mm
PROPERTY Position : LREAL
GET
Position := _Position.Position;
END_GET
SET
_Position.Position := Position;
END_SET
END_PROPERTY

//Registers Mover to be Monitored by Station
METHOD RegisterMover
VAR_INPUT
	Mover : I_XtsMover; //Mover to regsiter
END_VAR

VAR
	found	   : BOOL;
END_VAR
_RegisteredMovers.ResetIterator();
WHILE _RegisteredMovers.MoveToNext DO
	found := _RegisteredMovers.Current = Mover;
	IF found THEN
		RETURN;
	END_IF
END_WHILE

_RegisteredMovers.AddItem(Mover);
LogMessage.Message	 := CONCAT('Mover Registered: ', Mover.Name);
LogMessage.Severity	 := 0;
LogMessage.MessageId := E_XtsLogMessage.PositionTriggerGetMoverCalled;
_Logger.LogMessageInstance(LogSource, LogMessage);
END_METHOD

{attribute 'monitoring':='call'}
PROPERTY Status : I_XtsPositionTriggerStatus
GET
Status := _Status;
END_GET
END_PROPERTY

END_FUNCTION_BLOCK

// _Internal/PositionTrigger/Status/XtsPositionTriggerStatus
{attribute 'no_explicit_call' := 'This FB is a CLASS and must be accessed using methods or properties'}
FUNCTION_BLOCK XtsPositionTriggerStatus IMPLEMENTS I_XtsPositionTriggerStatus
VAR
	_PositionTrigger : I_XtsPositionTrigger;
	_Movers			 : I_XtsMoverCollection;
	_MonitorTask	 : I_MoverMonitor;
END_VAR

//FB_Init is always available implicitly and it is used primarily for initialization.

//The return value is not evaluated. For a specific influence, you can also declare the

//methods explicitly and provide additional code there with the standard initialization

//code. You can evaluate the return value.
METHOD FB_Init : BOOL
VAR_INPUT
	bInitRetains	: BOOL; // TRUE: the retain variables are initialized (reset warm / reset cold)
	bInCopyCode		: BOOL; // TRUE: the instance will be copied to the copy code afterward (online change)   
	PositionTrigger : I_XtsPositionTrigger;
	MonitorTask		: I_MoverMonitor;
END_VAR
_PositionTrigger := PositionTrigger;
_MonitorTask	 := MonitorTask;
END_METHOD

{attribute 'monitoring':='call'}
//Number of Movers Currently Registered to the Station
PROPERTY NumberOfMoverEvents : UDINT
GET
NumberOfMoverEvents := _PositionTrigger.MoverQueue.Count;
END_GET
END_PROPERTY

{attribute 'monitoring' := 'call'}
//Number of Movers Currently Registered to the Station
PROPERTY NumberOfMoversRegistered : UDINT
GET
NumberOfMoversRegistered := _Movers.Count;
END_GET
END_PROPERTY

METHOD SetRegisteredMovers
VAR_INPUT
	RegisteredMovers : I_XtsMoverCollection;
END_VAR
_Movers := RegisteredMovers;
END_METHOD

END_FUNCTION_BLOCK

// _Internal/Station/Interfaces/I_MoverMonitor
INTERFACE I_MoverMonitor EXTENDS I_Base, I_Cyclic

METHOD GetMover : I_XtsMover
VAR_INPUT
END_VAR
END_METHOD

PROPERTY MonitoredMovers : I_XtsMoverCollection
GET
END_GET
SET
END_SET
END_PROPERTY

{attribute 'monitoring':='call'}
PROPERTY MoverPresent : BOOL
GET
END_GET
END_PROPERTY

END_INTERFACE

// _Internal/Station/MoverThresholdMonitorTask
{attribute 'no_explicit_call' := 'This FB is a CLASS and must be accessed using methods or properties'}
FUNCTION_BLOCK MoverThresholdMonitorTask IMPLEMENTS I_MoverMonitor
VAR
	_MonitoredMovers : I_XtsMoverCollection;
	_MoverQueue		 : I_XtsMoverQueue;
	_CurrentMover	 : I_XtsMover := NullObjects.XtsMover;
	_Position		 : I_Positionable;
	_Logger			 : I_XtsLogger;
	LogSource		 : TraceSourceInfo;
	LogMessage		 : TraceMessageInfo;
END_VAR

METHOD CyclicLogic
VAR
	Mover				 : I_XtsMover;
	ThresholdEventResult : E_ThresholdEvent;
END_VAR
IF _MonitoredMovers = 0 THEN
	RETURN;
END_IF

_MonitoredMovers.ResetIterator();
WHILE _MonitoredMovers.MoveToNext DO
	__QUERYINTERFACE(_MonitoredMovers.Current, mover);
	ThresholdEventResult := CheckForThresholdEvent(Mover, _Position.Position);
	CASE ThresholdEventResult OF
		E_ThresholdEvent.NoEvent:
		//do nothing
		E_ThresholdEvent.PositiveEvent:
			LogMessage.MessageId := E_XtsLogMessage.PositionTriggerMoverPassedPositive;
			LogMessage.Message	 := CONCAT(Mover.Name, ' passed monitored position in positive direction');
			_Logger.LogMessageInstance(LogSource, LogMessage);
			_MoverQueue.Enqueue(mover);

		E_ThresholdEvent.NegativeEvent:
			LogMessage.MessageId := E_XtsLogMessage.PositionTriggerMoverPassedNegative;
			LogMessage.Message	 := CONCAT(Mover.Name, ' passed monitored position in negative direction');
			_MoverQueue.Enqueue(mover);
	END_CASE
END_WHILE
END_METHOD

//FB_Init is always available implicitly and it is used primarily for initialization.

//The return value is not evaluated. For a specific influence, you can also declare the

//methods explicitly and provide additional code there with the standard initialization

//code. You can evaluate the return value.
METHOD FB_Init : BOOL
VAR_INPUT
	bInitRetains	: BOOL; // TRUE: the retain variables are initialized (reset warm / reset cold)
	bInCopyCode		: BOOL; // TRUE: the instance will be copied to the copy code afterward (online change)
	PositionTrigger : I_XtsPositionTrigger;
END_VAR

VAR
	Queueable	  : I_Queueable;
END_VAR
__QUERYINTERFACE(PositionTrigger, _Position);
__QUERYINTERFACE(PositionTrigger, Queueable);
__QUERYINTERFACE(PositionTrigger.TracePublisher, _Logger);
_MoverQueue			 := Queueable.MoverQueue;
LogSource.SourceName := 'Threshold Monitor';
END_METHOD

METHOD GetMover : I_XtsMover
VAR
	
END_VAR
GetMover := NullObjects.XtsMover;
IF _MoverQueue.Count = 0 THEN
	LogMessage.Message	 := 'GetMover called when no mover present.';
	LogMessage.Severity	 := 2;
	LogMessage.MessageId := E_XtsLogMessage.StationGetMoverCalledNoMover;
	_Logger.LogMessageInstance(LogSource, LogMessage);
	RETURN;
END_IF

GetMover := _MoverQueue.Dequeue();
END_METHOD

PROPERTY MonitoredMovers : I_XtsMoverCollection
GET
MonitoredMovers := _MonitoredMovers;
END_GET
SET
_MonitoredMovers := MonitoredMovers;
END_SET
END_PROPERTY

{attribute 'monitoring':='call'}
PROPERTY MoverPresent : BOOL
GET
MoverPresent := _MoverQueue.Count > 0;
END_GET
END_PROPERTY

METHOD SetMonitoredMovers
VAR_INPUT
	Movers : I_XtsMoverCollection;
END_VAR
_MonitoredMovers := Movers;
END_METHOD

END_FUNCTION_BLOCK

// _Internal/Station/CheckForThresholdEvent
FUNCTION CheckForThresholdEvent : E_ThresholdEvent
VAR_INPUT
	Mover			  : I_XtsMover;
	ThresholdPosition : LREAL;
END_VAR

VAR_STAT
	track				: I_XtsTrack;
	lastCyclePosition	: LREAL;
	normalizedCurrent	: LREAL;
	normalizedThreshold : LREAL;
END_VAR

CheckForThresholdEvent := E_ThresholdEvent.NoEvent;
track				   := Mover.Status.CurrentTrack;
lastCyclePosition	   := Mover.LastCyclePosition;
normalizedCurrent	   := Mover.Position;
normalizedThreshold	   := MODABS(ThresholdPosition, track.Length);
// Unwrap current position relative to last position
IF (normalizedCurrent - lastCyclePosition) > (track.Length / 2.0) THEN
	normalizedCurrent := normalizedCurrent - track.Length;
ELSIF (normalizedCurrent - lastCyclePosition) < -(track.Length / 2.0) THEN
	normalizedCurrent := normalizedCurrent + track.Length;
END_IF;

// Unwrap threshold relative to last position
IF (normalizedThreshold - lastCyclePosition) > (track.Length / 2.0) THEN
	normalizedThreshold := normalizedThreshold - track.Length;
ELSIF (normalizedThreshold - lastCyclePosition) < -(track.Length / 2.0) THEN
	normalizedThreshold := normalizedThreshold + track.Length;
END_IF;

// Now simple linear comparison works
IF lastCyclePosition < normalizedThreshold AND normalizedCurrent >= normalizedThreshold THEN
	CheckForThresholdEvent := E_ThresholdEvent.PositiveEvent;
ELSIF lastCyclePosition > normalizedThreshold AND normalizedCurrent <= normalizedThreshold THEN
	CheckForThresholdEvent := E_ThresholdEvent.NegativeEvent;
END_IF;

END_FUNCTION

// _Internal/NullObjects/NullStation
{attribute 'no_explicit_call' := 'This FB is a CLASS and must be accessed using methods or properties'}
{attribute 'conditionalshow'}
{warning disable C0094}
{warning disable C0568}
FUNCTION_BLOCK NullStation EXTENDS CyclicComponent IMPLEMENTS I_XtsStation, I_NullObject
VAR
END_VAR

METHOD AcceptStationVisitor
VAR_INPUT
	StationVisitor : I_XtsStationVisitor;
END_VAR
END_METHOD

{attribute 'monitoring':='call'}
PROPERTY CommandLog : I_XtsLocalLog
GET
CommandLog := NullObjects.MechatronicsLocalLog;
END_GET
END_PROPERTY

METHOD CyclicLogic
END_METHOD

METHOD DeregisterMover
VAR_INPUT
	Mover : I_XtsMover;
END_VAR
END_METHOD

METHOD Disable
END_METHOD

METHOD Enable
END_METHOD

PROPERTY Enabled : BOOL
GET
END_GET
END_PROPERTY

METHOD GetMover : I_XtsMover
GetMover := NullObjects.XtsMover;
END_METHOD

METHOD IsMoverRegistered : BOOL
VAR_INPUT
	Mover : I_XtsMover;
END_VAR
END_METHOD

PROPERTY MoverIsPresent : BOOL
GET
END_GET
END_PROPERTY

PROPERTY Movers : I_XtsMoverEnumerator
GET
Movers := NullObjects.MoverCollection;
END_GET
END_PROPERTY

PROPERTY Position : LREAL
GET
END_GET
SET
END_SET
END_PROPERTY

METHOD RegisterMover
VAR_INPUT
	Mover	: I_XtsMover;
END_VAR
END_METHOD

{attribute 'monitoring':='call'}
PROPERTY Status : I_XtsStationStatus
GET
Status := NullObjects.XtsStationStatus;
END_GET
END_PROPERTY

PROPERTY TracePublisher : I_XtsTracePublisher
GET
TracePublisher := NullObjects.MechatronicsTracePublisher;
END_GET
END_PROPERTY

END_FUNCTION_BLOCK

// _Internal/Station/Status/XtsStationStatus
{attribute 'no_explicit_call' := 'This FB is a CLASS and must be accessed using methods or properties'}
FUNCTION_BLOCK XtsStationStatus IMPLEMENTS I_XtsStationStatus
VAR
	_Station	 : I_XtsStation;
	_Movers		 : I_XtsMoverCollection;
	_MonitorTask : I_MoverMonitor;
END_VAR

//FB_Init is always available implicitly and it is used primarily for initialization.

//The return value is not evaluated. For a specific influence, you can also declare the

//methods explicitly and provide additional code there with the standard initialization

//code. You can evaluate the return value.
METHOD FB_Init : BOOL
VAR_INPUT
	bInitRetains : BOOL; // TRUE: the retain variables are initialized (reset warm / reset cold)
	bInCopyCode	 : BOOL; // TRUE: the instance will be copied to the copy code afterward (online change)   
	Station		 : I_XtsStation;
	MonitorTask	 : I_MoverMonitor;
END_VAR
_Station	 := Station;
_MonitorTask := MonitorTask;
END_METHOD

{attribute 'monitoring' := 'call'}
//Number of Movers Currently Registered to the Station
PROPERTY NumberOfMoversRegistered : UDINT
GET
NumberOfMoversRegistered := _Movers.Count;
END_GET
END_PROPERTY

METHOD SetRegisteredMovers
VAR_INPUT
	RegisteredMovers : I_XtsMoverCollection;
END_VAR
_Movers := RegisteredMovers;
END_METHOD

END_FUNCTION_BLOCK

// _Internal/NullObjects/NullStationCollection
{attribute 'no_explicit_call' := 'This FB is a CLASS and must be accessed using methods or properties'}
{attribute 'conditionalshow'}
{warning disable C0094}
{warning disable C0568}
FUNCTION_BLOCK NullStationCollection IMPLEMENTS I_XtsStationCollection, I_NullObject
VAR
END_VAR

METHOD AcceptStationVisitor
VAR_INPUT
	StationVisitor : I_XtsStationVisitor;
END_VAR
END_METHOD

METHOD AddItem
VAR_INPUT
	Station	: I_XtsStation;
END_VAR
END_METHOD

METHOD Clear
END_METHOD

PROPERTY Count : UDINT
GET
END_GET
END_PROPERTY

PROPERTY Current : I_XtsStation
GET
Current := NullObjects.Station;
END_GET
END_PROPERTY

PROPERTY CurrentItem : UDINT
GET
END_GET
END_PROPERTY

PROPERTY IsEmpty : BOOL
GET
END_GET
END_PROPERTY

PROPERTY MoveToNext : BOOL
GET
END_GET
END_PROPERTY

METHOD Remove
VAR_INPUT
	Station	: I_XtsStation;
END_VAR
END_METHOD

METHOD ResetIterator
END_METHOD

END_FUNCTION_BLOCK

// _Internal/NullObjects/NullSyncAxisParameters
{attribute 'no_explicit_call' := 'This FB is a CLASS and must be accessed using methods or properties'}
{attribute 'conditionalshow'}
{warning disable C0094}
FUNCTION_BLOCK NullSyncAxisParameters IMPLEMENTS I_SyncAxisParameters, I_NullObject
VAR
END_VAR

{attribute 'monitoring':='call'}
PROPERTY MasterAxis : REFERENCE TO AXIS_REF
GET
END_GET
SET
END_SET
END_PROPERTY

{attribute 'monitoring' := 'call'}
PROPERTY MasterStartDistance : MC_LREAL
GET
END_GET
SET
END_SET
END_PROPERTY

{attribute 'monitoring' := 'call'}
PROPERTY MasterSyncPosition : MC_LREAL
GET
END_GET
SET
END_SET
END_PROPERTY

PROPERTY Options_CA : REFERENCE TO Tc3_McCollisionAvoidance.ST_GearInPosCAOptions
GET
END_GET
SET
END_SET
END_PROPERTY

{attribute 'monitoring' := 'call'}
PROPERTY RatioDenominator : UINT
GET
END_GET
SET
END_SET
END_PROPERTY

{attribute 'monitoring' := 'call'}
PROPERTY RatioNumerator : MC_LREAL
GET
END_GET
SET
END_SET
END_PROPERTY

{attribute 'monitoring' := 'call'}
PROPERTY SlaveSyncPosition : LREAL
GET
END_GET
SET
END_SET
END_PROPERTY

{attribute 'monitoring' := 'call'}
PROPERTY SyncMode : Tc3_McCollisionAvoidance.MC_SYNC_MODE
GET
END_GET
SET
END_SET
END_PROPERTY

{attribute 'monitoring' := 'call'}
PROPERTY SyncStrategy : Tc3_McCollisionAvoidance.MC_SYNC_STRATEGY
GET
END_GET
SET
END_SET
END_PROPERTY

END_FUNCTION_BLOCK

// _Internal/NullObjects/NullXtsModule
{attribute 'no_explicit_call' := 'This FB is a CLASS and must be accessed using methods or properties'}
{attribute 'conditionalshow'}
{warning disable C0094}
{warning disable C0568}
FUNCTION_BLOCK NullXtsModule EXTENDS CyclicComponent IMPLEMENTS I_XtsModule, I_NullObject
VAR
END_VAR

METHOD Accept
VAR_INPUT
	ComponentVisitor	: Core.I_ComponentVisitor;
END_VAR
END_METHOD

METHOD AcceptXtsModuleVisitor
VAR_INPUT
	XtsModuleVisitor : I_XtsModuleVisitor;
END_VAR
END_METHOD

PROPERTY CurveAngle : LREAL
GET
END_GET
END_PROPERTY

METHOD CyclicLogic
END_METHOD

METHOD Dispose
END_METHOD

PROPERTY Gap : LREAL
GET
END_GET
END_PROPERTY

PROPERTY HMI : I_HmiFunction
GET
END_GET
END_PROPERTY

PROPERTY Id : UDINT
GET
END_GET
SET
END_SET
END_PROPERTY

METHOD Initialize
END_METHOD

{attribute 'monitoring' := 'call'}
PROPERTY Initialized : BOOL
GET
END_GET
SET
END_SET
END_PROPERTY

PROPERTY Length : LREAL
GET
END_GET
END_PROPERTY

{attribute 'monitoring':='call'}
PROPERTY Module24Vdc : REAL
GET
END_GET
END_PROPERTY

{attribute 'monitoring':='call'}
PROPERTY Module48Vdc : REAL
GET
END_GET
END_PROPERTY

{attribute 'monitoring':='call'}
PROPERTY ModuleReady : BOOL
GET
END_GET
END_PROPERTY

{attribute 'monitoring' := 'call'}
PROPERTY Name : Core.T_MaxString
GET
END_GET
SET
END_SET
END_PROPERTY

{attribute 'monitoring':='call'}
PROPERTY Otcid : OTCID
GET
END_GET
SET
END_SET
END_PROPERTY

METHOD RegisterWithParent
VAR_INPUT
	Parent	: Core.I_ContainComponents;
END_VAR
END_METHOD

PROPERTY Utility : I_TcIoXtsPartModule
GET
END_GET
SET
END_SET
END_PROPERTY

PROPERTY Vdc24Okay : BOOL
GET
END_GET
END_PROPERTY

PROPERTY Vdc48Okay : BOOL
GET
END_GET
END_PROPERTY

PROPERTY XtsModuleType : Tc3_Xts_Utility.ModuleType
GET
END_GET
END_PROPERTY

END_FUNCTION_BLOCK

// _Internal/NullObjects/NullXtsModuleCollection
{attribute 'no_explicit_call' := 'This FB is a CLASS and must be accessed using methods or properties'}
{attribute 'conditionalshow'}
{warning disable C0094}
FUNCTION_BLOCK NullXtsModuleCollection IMPLEMENTS I_XtsModuleCollection, I_NullObject
VAR
END_VAR

METHOD Clear
END_METHOD

{attribute 'monitoring' := 'call'}
PROPERTY Count : UDINT
GET
END_GET
END_PROPERTY

METHOD Create : BOOL
VAR_INPUT
	NumberOfModules	: UINT;
END_VAR
END_METHOD

{attribute 'monitoring':='call'}
PROPERTY Current : I_XtsModule
GET
Current := NullObjects.XtsModule;
END_GET
END_PROPERTY

{attribute 'monitoring' := 'call'}
PROPERTY CurrentItem : UDINT
GET
END_GET
END_PROPERTY

METHOD Dispose
END_METHOD

METHOD GetById : I_XtsModule
VAR_INPUT
	ModuleId	: UDINT;
END_VAR
GetById := NullObjects.XtsModule;
END_METHOD

METHOD GetByOtcid : I_XtsModule
VAR_INPUT
	ModuleOtcid	: OTCID;
END_VAR
GetByOtcid := NullObjects.XtsModule;
END_METHOD

{attribute 'monitoring' := 'call'}
PROPERTY IsEmpty : BOOL
GET
END_GET
END_PROPERTY

PROPERTY MoveToNext : BOOL
GET
END_GET
END_PROPERTY

METHOD ResetIterator
END_METHOD

END_FUNCTION_BLOCK

// _Internal/NullObjects/NullXtsMover
{attribute 'no_explicit_call' := 'This FB is a CLASS and must be accessed using methods or properties'}
{attribute 'conditionalshow'}
{warning disable C0094}
{warning disable C0568}
FUNCTION_BLOCK NullXtsMover IMPLEMENTS I_XtsMover, I_NullObject
VAR
END_VAR

METHOD Accept
VAR_INPUT
	ComponentVisitor	: Core.I_ComponentVisitor;
END_VAR
END_METHOD

METHOD AcceptMoverVisitor
VAR_INPUT
	MoverVisitor : I_XtsMoverVisitor;
END_VAR
END_METHOD

METHOD ActivateTrack : I_XtsMoverTaskResult
VAR_INPUT
	TrackId	: UDINT;
END_VAR
ActivateTrack := NullObjects.XtsMoverTask;
END_METHOD

METHOD AddToGroup : I_XtsMoverTaskResult
VAR_INPUT
	Group	: REFERENCE TO AXES_GROUP_REF;
	Ident	: UDINT;
END_VAR
AddToGroup := NullObjects.XtsMoverTask;
END_METHOD

PROPERTY Axis : REFERENCE TO Tc2_MC2.AXIS_REF
GET
END_GET
END_PROPERTY

{attribute 'monitoring' := 'call'}
PROPERTY Busy : BOOL
GET
END_GET
END_PROPERTY

{attribute 'monitoring':='call'}
PROPERTY CommandLog : I_XtsLocalLog
GET
CommandLog := NullObjects.MechatronicsLocalLog;
END_GET
END_PROPERTY

PROPERTY CurrentTask : I_XtsMoverTaskResult
GET
CurrentTask := NullObjects.XtsMoverTask;
END_GET
END_PROPERTY

METHOD DeregisterWithParent
VAR_INPUT
	Parent	: Core.I_ContainComponents;
END_VAR
END_METHOD

METHOD Disable
END_METHOD

METHOD Enable
END_METHOD

PROPERTY Enabled : BOOL
GET
END_GET
END_PROPERTY

{attribute 'monitoring' := 'call'}
PROPERTY Error : BOOL
GET
END_GET
END_PROPERTY

{attribute 'monitoring' := 'call'}
PROPERTY ErrorId : UDINT
GET
END_GET
END_PROPERTY

METHOD Halt : I_XtsMoverTaskResult
VAR_INPUT
	Deceleration	: LREAL;
	Gap	: LREAL;
END_VAR
Halt := NullObjects.XtsMoverTask;
END_METHOD

METHOD Initialize
END_METHOD

{attribute 'monitoring' := 'call'}
PROPERTY Initialized : BOOL
GET
END_GET
SET
END_SET
END_PROPERTY

PROPERTY InPosition : BOOL
GET
END_GET
END_PROPERTY

PROPERTY InVelocity : BOOL
GET
END_GET
END_PROPERTY

PROPERTY LastCyclePosition : LREAL
GET
END_GET
END_PROPERTY

{attribute 'monitoring':='call'}
PROPERTY ManualGroupControl : BOOL
GET
END_GET
SET
END_SET
END_PROPERTY

{attribute 'monitoring':='call'}
PROPERTY MoverData : I_XtsMoverData
GET
MoverData := NullObjects.XtsMoverData;
END_GET
SET
END_SET
END_PROPERTY

{attribute 'monitoring':='call'}
PROPERTY MoverId : UDINT
GET
END_GET
END_PROPERTY

PROPERTY MoverTasks : I_XtsMoverTaskCollection
GET
MoverTasks := NullObjects.XtsMoverTaskCollection;
END_GET
END_PROPERTY

PROPERTY MoverUtility : I_TcIoXtsXpuMover
GET
END_GET
SET
END_SET
END_PROPERTY

METHOD MoveToPosition : I_XtsMoverTaskResult
VAR_INPUT
	Position	: LREAL;
	Direction	: Tc3_Mc3Definitions.MC_DIRECTION := .Tc3_Mc3Definitions.MC_DIRECTION.mcDirectionPositive;
END_VAR
MoveToPosition := NullObjects.XtsMoverTask;
END_METHOD

METHOD MoveToStation : I_XtsMoverTaskResult
VAR_INPUT
	Station	: I_XtsStation;
END_VAR
MoveToStation := NullObjects.XtsMoverTask;
END_METHOD

METHOD MoveVelocity : I_XtsMoverTaskResult
VAR_INPUT
	Velocity	: LREAL;
	Direction	: Tc3_Mc3Definitions.MC_DIRECTION := .Tc3_Mc3Definitions.MC_DIRECTION.mcDirectionPositive;
END_VAR
MoveVelocity := NullObjects.XtsMoverTask;
END_METHOD

PROPERTY Name : Core.T_MaxString
GET
Name := 'Null Mover';
END_GET
SET
END_SET
END_PROPERTY

PROPERTY Parameters : I_XtsParameterSet
GET
Parameters := NullObjects.XtsParameterSet;
END_GET
SET
END_SET
END_PROPERTY

PROPERTY Position : LREAL
GET
END_GET
END_PROPERTY

METHOD RefreshMoverId
VAR_INPUT
	Xpu	: I_TcIoXtsProcessingUnit;
END_VAR
END_METHOD

METHOD RegisterWithParent
VAR_INPUT
	Parent	: Core.I_ContainComponents;
END_VAR
END_METHOD

METHOD RemoveFromGroup : I_XtsMoverTaskResult
VAR_INPUT
	Group	: REFERENCE TO AXES_GROUP_REF;
	Ident	: UDINT;
END_VAR
RemoveFromGroup := NullObjects.XtsMoverTask;
END_METHOD

METHOD Reset
END_METHOD

PROPERTY Status : I_XtsMoverStatus
GET
Status := NullObjects.XtsMoverStatus;
END_GET
END_PROPERTY

METHOD SyncToAxis : I_XtsMoverTaskResult
VAR_INPUT
	Master			   : REFERENCE TO AXIS_REF;
	MasterSyncPosition : LREAL;
	SlaveSyncPosition  : LREAL;
END_VAR
SyncToAxis := NullObjects.XtsMoverTask;
END_METHOD

METHOD SyncToMover : I_XtsMoverTaskResult
VAR_INPUT
	Master	 : I_XtsMover;
	Distance : LREAL;
END_VAR
SyncToMover := NullObjects.XtsMoverTask;
END_METHOD

PROPERTY TracePublisher : I_XtsTracePublisher
GET
TracePublisher := NullObjects.MechatronicsTracePublisher;
END_GET
END_PROPERTY

PROPERTY Tracks : I_XtsTrackCollection
GET
Tracks := NullObjects.XtsTrackCollection;
END_GET
SET
END_SET
END_PROPERTY

{attribute 'monitoring':='call'}
PROPERTY VirtualMover : BOOL
GET
END_GET
SET
END_SET
END_PROPERTY

END_FUNCTION_BLOCK

// _Internal/NullObjects/NullXtsMoverData
{attribute 'no_explicit_call' := 'This FB is a CLASS and must be accessed using methods or properties'}
{attribute 'conditionalshow'}
{warning disable C0094}
FUNCTION_BLOCK NullXtsMoverData IMPLEMENTS I_XtsMoverData, I_NullObject
VAR
END_VAR

END_FUNCTION_BLOCK

// _Internal/NullObjects/NullXtsMoverList
{attribute 'no_explicit_call' := 'This FB is a CLASS and must be accessed using methods or properties'}
{attribute 'conditionalshow'}
{warning disable C0094}
{warning disable C0568}
FUNCTION_BLOCK NullXtsMoverList IMPLEMENTS I_XtsMoverList, I_NullObject
VAR
END_VAR

METHOD AcceptMoverVisitor
VAR_INPUT
	MoverVisitor : I_XtsMoverVisitor;
END_VAR
END_METHOD

METHOD AddItem
VAR_INPUT
	Mover	: I_XtsMover;
END_VAR
END_METHOD

METHOD Clear
END_METHOD

METHOD Contains : BOOL
VAR_INPUT
	Mover	: I_XtsMover;
END_VAR
END_METHOD

{attribute 'monitoring' := 'call'}
PROPERTY Count : UDINT
GET
END_GET
END_PROPERTY

PROPERTY Current : I_XtsMover
GET
Current := NullObjects.XtsMover;
END_GET
END_PROPERTY

PROPERTY CurrentItem : UDINT
GET
END_GET
END_PROPERTY

METHOD GetAtIndex : I_XtsMover
VAR_INPUT
	Index	: UDINT;
END_VAR
GetAtIndex := NullObjects.XtsMover;
END_METHOD

METHOD InsertAtIndex
VAR_INPUT
	Mover	: I_XtsMover;
	Index	: UDINT;
END_VAR
END_METHOD

PROPERTY IsEmpty : BOOL
GET
END_GET
END_PROPERTY

METHOD Map
VAR_INPUT
	Validator : I_XtsMoverValidator;
	Visitor	  : I_XtsMoverVisitor;
END_VAR
END_METHOD

PROPERTY Mover : UDINT
GET
END_GET
END_PROPERTY

PROPERTY MoveToNext : BOOL
GET
END_GET
END_PROPERTY

METHOD Remove
VAR_INPUT
	Mover	: I_XtsMover;
END_VAR
END_METHOD

METHOD RemoveAtIndex
VAR_INPUT
	MoverIndex	: UDINT;
END_VAR
END_METHOD

METHOD ResetIterator
END_METHOD

END_FUNCTION_BLOCK

// _Internal/NullObjects/NullXtsMoverStatus
{attribute 'no_explicit_call' := 'This FB is a CLASS and must be accessed using methods or properties'}
{attribute 'conditionalshow'}
{warning disable C0094}
FUNCTION_BLOCK NullXtsMoverStatus IMPLEMENTS I_XtsMoverStatus, I_NullObject
VAR
END_VAR

{attribute 'monitoring':='call'}
PROPERTY ActualAcceleration : LREAL
GET
END_GET
END_PROPERTY

{attribute 'monitoring':='call'}
PROPERTY ActualVelocity : LREAL
GET
END_GET
END_PROPERTY

{attribute 'monitoring':='call'}
PROPERTY AvoidingCollision : BOOL
GET
END_GET
END_PROPERTY

{attribute 'monitoring' := 'call'}
PROPERTY Axis : I_AxisRef
GET
Axis := NullObjects.Axis;
END_GET
END_PROPERTY

{attribute 'monitoring' := 'call'}
PROPERTY CommandedPosition : LREAL
GET
END_GET
SET
END_SET
END_PROPERTY

{attribute 'monitoring':='call'}
PROPERTY CommandedStation : I_XtsStation
GET
END_GET
SET
END_SET
END_PROPERTY

{attribute 'monitoring' := 'call'}
PROPERTY CurrentStation : I_Station
GET
CurrentStation := NullObjects.Station;
END_GET
END_PROPERTY

{attribute 'monitoring' := 'call'}
PROPERTY CurrentTrack : I_XtsTrack
GET
CurrentTrack := NullObjects.XtsTrack;
END_GET
SET
END_SET
END_PROPERTY

{attribute 'monitoring':='call'}
PROPERTY IdentInGroup : UDINT
GET
END_GET
SET
END_SET
END_PROPERTY

{attribute 'monitoring' := 'call'}
PROPERTY InSync : BOOL
GET
END_GET
SET
END_SET
END_PROPERTY

{attribute 'monitoring':='call'}
PROPERTY MoverInGroup : BOOL
GET
END_GET
END_PROPERTY

{attribute 'monitoring':='call'}
PROPERTY SetAcceleration : LREAL
GET
END_GET
END_PROPERTY

{attribute 'monitoring' := 'call'}
PROPERTY SetVelocity : LREAL
GET
END_GET
END_PROPERTY

END_FUNCTION_BLOCK

// _Internal/NullObjects/NullXtsMoverTaskCollection
{attribute 'no_explicit_call' := 'This FB is a CLASS and must be accessed using methods or properties'}
{attribute 'conditionalshow'}
{warning disable C0094}
FUNCTION_BLOCK NullXtsMoverTaskCollection IMPLEMENTS I_XtsMoverTaskCollection, I_NullObject
VAR
END_VAR

METHOD AddTask : BOOL
VAR_INPUT
	Task	: I_XtsMoverTask;
END_VAR
END_METHOD

PROPERTY ErrorTask : T_MaxString
GET
END_GET
END_PROPERTY

METHOD GetTaskById : I_XtsMoverTask
VAR_INPUT
	TaskId	: MoverTaskID;
END_VAR
GetTaskById := NullObjects.XtsMoverTask;
END_METHOD

METHOD GetTaskByName : I_XtsMoverTask
VAR_INPUT
	Name	: T_MaxString;
END_VAR
GetTaskByName := NullObjects.XtsMoverTask;
END_METHOD

METHOD RemoveTaskById : BOOL
VAR_INPUT
	TaskId	: MoverTaskId;
END_VAR
END_METHOD

METHOD RemoveTaskByInstance : BOOL
VAR_INPUT
	Task	: I_XtsMoverTask;
END_VAR
END_METHOD

END_FUNCTION_BLOCK

// _Internal/NullObjects/NullXtsMoverTaskResult
{attribute 'no_explicit_call' := 'This FB is a CLASS and must be accessed using methods or properties'}
{attribute 'conditionalshow'}
{warning disable C0094}
{warning disable C0568}
FUNCTION_BLOCK NullXtsMoverTaskResult IMPLEMENTS I_XtsMoverTaskResult, I_NullObject
VAR
END_VAR

PROPERTY Aborted : BOOL
GET
END_GET
END_PROPERTY

PROPERTY Busy : BOOL
GET
END_GET
END_PROPERTY

PROPERTY CommandExecuted : BOOL
GET
END_GET
END_PROPERTY

PROPERTY Error : BOOL
GET
END_GET
END_PROPERTY

PROPERTY ErrorId : UDINT
GET
END_GET
END_PROPERTY

PROPERTY TaskId : MoverTaskId
GET
END_GET
END_PROPERTY

PROPERTY TaskName : STRING
GET
TaskName := 'Null Xts Mover Task';
END_GET
END_PROPERTY

END_FUNCTION_BLOCK

// _Internal/NullObjects/NullXtsParameterSet
{attribute 'no_explicit_call' := 'This FB is a CLASS and must be accessed using methods or properties'}
{attribute 'conditionalshow'}
{warning disable C0094}
{warning disable C0568}
FUNCTION_BLOCK NullXtsParameterSet IMPLEMENTS I_XtsParameterSet, I_NullObject
VAR
	_NullXtsTrack		: NullXtsTrack;
	_NullXtsStation		: NullStation('Null Xts Station');
	_SyncAxisParameters : NullSyncAxisParameters;
END_VAR

PROPERTY Acceleration : LREAL
GET
END_GET
SET
END_SET
END_PROPERTY

METHOD CopyFrom
VAR_INPUT
	Other	: I_XtsParameterSet;
END_VAR
END_METHOD

METHOD CopyTo
VAR_INPUT
	Other	: I_XtsParameterSet;
END_VAR
END_METHOD

PROPERTY Deceleration : LREAL
GET
END_GET
SET
END_SET
END_PROPERTY

PROPERTY Direction : Tc3_Mc3Definitions.MC_DIRECTION
GET
END_GET
SET
END_SET
END_PROPERTY

PROPERTY Gap : LREAL
GET
END_GET
SET
END_SET
END_PROPERTY

PROPERTY Jerk : LREAL
GET
END_GET
SET
END_SET
END_PROPERTY

PROPERTY Position : LREAL
GET
END_GET
SET
END_SET
END_PROPERTY

{attribute 'monitoring':='call'}
PROPERTY SyncAxis : I_SyncAxisParameters
GET
SyncAxis := NullObjects.SyncAxisParameters;
END_GET
END_PROPERTY

PROPERTY Track : I_XtsTrack
GET
Track := NullObjects.XtsTrack;
END_GET
SET
END_SET
END_PROPERTY

PROPERTY Velocity : LREAL
GET
END_GET
SET
END_SET
END_PROPERTY

END_FUNCTION_BLOCK

// _Internal/NullObjects/NullXtsTrack
{attribute 'no_explicit_call' := 'This FB is a CLASS and must be accessed using methods or properties'}
{attribute 'conditionalshow'}
{warning disable C0094}
{warning disable C0568}
FUNCTION_BLOCK NullXtsTrack IMPLEMENTS I_XtsTrack, I_NullObject
VAR
END_VAR

METHOD Dispose
END_METHOD

PROPERTY Id : UDINT
GET
Id := 65535;
END_GET
SET
END_SET
END_PROPERTY

PROPERTY Length : LREAL
GET
END_GET
SET
END_SET
END_PROPERTY

PROPERTY Offset : LREAL
GET
END_GET
SET
END_SET
END_PROPERTY

PROPERTY Otcid : OTCID
GET
END_GET
SET
END_SET
END_PROPERTY

PROPERTY Polarity : Polarity
GET
END_GET
SET
END_SET
END_PROPERTY

PROPERTY Utility : I_TcIoXtsXpuTrack
GET
END_GET
SET
END_SET
END_PROPERTY

END_FUNCTION_BLOCK

// _Internal/NullObjects/NullXtsPart
{attribute 'no_explicit_call' := 'This FB is a CLASS and must be accessed using methods or properties'}
{attribute 'conditionalshow'}
{warning disable C0094}
{warning disable C0568}
FUNCTION_BLOCK NullXtsPart IMPLEMENTS I_XtsPart, I_NullObject
VAR
END_VAR

METHOD Accept
VAR_INPUT
	Visitor	: Core.I_ModuleVisitor;
END_VAR
END_METHOD

METHOD AcceptXtsModuleVisitor
VAR_INPUT
	XtsModuleVisitor : I_XtsModuleVisitor;
END_VAR
END_METHOD

METHOD AcceptXtsPartVisitor
VAR_INPUT
	XtsPartVisitor : I_XtsPartVisitor;
END_VAR
END_METHOD

PROPERTY Components : Core.I_ComponentCollection
GET
END_GET
END_PROPERTY

METHOD CyclicLogic
END_METHOD

METHOD DeregisterComponent : RegistrationResult
VAR_INPUT
	Component	: I_Component;
END_VAR
END_METHOD

METHOD DeregisterCyclic : RegistrationResult
VAR_INPUT
	Cyclic	: I_Cyclic;
END_VAR
END_METHOD

METHOD DeregisterInitialize : RegistrationResult
VAR_INPUT
	Initializable	: Core.I_Initializable;
END_VAR
END_METHOD

METHOD DeregisterModule : RegistrationResult
VAR_INPUT
	Module	: Core.I_Module;
END_VAR
END_METHOD

METHOD DeregisterWithParent 
VAR_INPUT
	Parent	: Core.I_ContainModules;
END_VAR
END_METHOD

METHOD Dispose
END_METHOD

PROPERTY Id : UDINT
GET
END_GET
SET
END_SET
END_PROPERTY

METHOD Initialize
END_METHOD

PROPERTY Initialized : BOOL
GET
END_GET
SET
END_SET
END_PROPERTY

PROPERTY Modules : I_ModuleCollection
GET
END_GET
END_PROPERTY

PROPERTY Name : Core.T_MaxString
GET
Name := 'Null Xts Part';
END_GET
END_PROPERTY

{attribute 'monitoring':='call'}
PROPERTY NumberModulesNotReady : UINT
GET
END_GET
END_PROPERTY

{attribute 'monitoring':='call'}
PROPERTY NumberModulesReady : UINT
GET
END_GET
END_PROPERTY

PROPERTY PartReady : BOOL
GET
END_GET
END_PROPERTY

PROPERTY Properties : I_XtsPartProperties
GET
END_GET
END_PROPERTY

METHOD RegisterComponent : RegistrationResult
VAR_INPUT
	Component	: Core.I_Component;
END_VAR
END_METHOD

METHOD RegisterCyclic : RegistrationResult
VAR_INPUT
	Cyclic	: Core.I_Cyclic;
END_VAR
END_METHOD

METHOD RegisterInitialize : RegistrationResult
VAR_INPUT
	Initializable	: Core.I_Initializable;
END_VAR
END_METHOD

METHOD RegisterModule : RegistrationResult
VAR_INPUT
	Module	: Core.I_Module;
END_VAR
END_METHOD

METHOD RegisterWithParent
VAR_INPUT
	Parent	: Core.I_ContainModules;
END_VAR
END_METHOD

METHOD ResetComponents : BOOL
END_METHOD

METHOD ResetModules : BOOL
END_METHOD

PROPERTY Utility : I_TcIoXtsXpuPart
GET
END_GET
SET
END_SET
END_PROPERTY

PROPERTY Vdc24Okay : BOOL
GET
END_GET
END_PROPERTY

PROPERTY Vdc48Okay : BOOL
GET
END_GET
END_PROPERTY

PROPERTY XtsModules : I_XtsModuleCollection
GET
XtsModules := NullObjects.XtsModuleCollection;
END_GET
END_PROPERTY

PROPERTY XtsPartId : UINT
GET
END_GET
SET
END_SET
END_PROPERTY

END_FUNCTION_BLOCK

// _Internal/NullObjects/NullXtsPartCollection
{attribute 'no_explicit_call' := 'This FB is a CLASS and must be accessed using methods or properties'}
{attribute 'conditionalshow'}
{warning disable C0094}
FUNCTION_BLOCK NullXtsPartCollection IMPLEMENTS I_XtsPartCollection, I_NullObject
VAR
END_VAR

METHOD AddItem
VAR_INPUT
	Part : I_XtsPart;
END_VAR
END_METHOD

METHOD Clear
VAR_INPUT
END_VAR
END_METHOD

{attribute 'monitoring' := 'call'}
PROPERTY Count : UDINT
GET
END_GET
END_PROPERTY

{attribute 'monitoring':='call'}
PROPERTY Current : I_XtsPart
GET
Current := NullObjects.XtsPart;
END_GET
END_PROPERTY

{attribute 'monitoring' := 'call'}
PROPERTY CurrentItem : UDINT
GET
END_GET
END_PROPERTY

METHOD GetById : I_XtsPart
VAR_INPUT
	PartId : UDINT;
END_VAR
GetById := NullObjects.XtsPart;
END_METHOD

METHOD GetByOtcid : I_XtsPart
VAR_INPUT
	PartOtcid : OTCID;
END_VAR
GetByOtcid := NullObjects.XtsPart;
END_METHOD

{attribute 'monitoring' := 'call'}
PROPERTY IsEmpty : BOOL
GET
END_GET
END_PROPERTY

PROPERTY MoveToNext : BOOL
GET
END_GET
END_PROPERTY

METHOD Remove
VAR_INPUT
	Part : I_XtsPart;
END_VAR
END_METHOD

METHOD ResetIterator
END_METHOD

END_FUNCTION_BLOCK

// _Internal/NullObjects/NullXtsPartTask
{attribute 'no_explicit_call' := 'This FB is a CLASS and must be accessed using methods or properties'}
FUNCTION_BLOCK NullXtsPartTask IMPLEMENTS I_XtsPartTask, I_NullObject

{attribute 'monitoring' := 'call'}
PROPERTY Busy : BOOL
GET
END_GET
END_PROPERTY

{attribute 'monitoring' := 'call'}
PROPERTY Error : BOOL
GET
END_GET
END_PROPERTY

{attribute 'monitoring' := 'call'}
PROPERTY ErrorId : UDINT
GET
END_GET
END_PROPERTY

{attribute 'monitoring':='call'}
PROPERTY TaskName : STRING
GET
TaskName := 'Null Xts Part Task';
END_GET
END_PROPERTY

PROPERTY XtsPartId : I_XtsPartId
GET
END_GET
SET
END_SET
END_PROPERTY

END_FUNCTION_BLOCK

// _Internal/NullObjects/NullXtsPositionTrigger
{attribute 'no_explicit_call' := 'This FB is a CLASS and must be accessed using methods or properties'}
{attribute 'conditionalshow'}
{warning disable C0094}
{warning disable C0568}
FUNCTION_BLOCK NullXtsPositionTrigger IMPLEMENTS I_XtsPositionTrigger, I_NullObject
VAR
END_VAR

METHOD Accept
VAR_INPUT
	ComponentVisitor	: Core.I_ComponentVisitor;
END_VAR
END_METHOD

METHOD AcceptXtsPositionTriggerVisitor
VAR_INPUT
	PositionTriggerVisitor : I_VisitXtsPositionTrigger;
END_VAR
END_METHOD

{attribute 'monitoring':='call'}
PROPERTY CommandLog : I_XtsLocalLog
GET
CommandLog := NullObjects.MechatronicsLocalLog;
END_GET
END_PROPERTY

METHOD DeregisterMover
VAR_INPUT
	Mover : I_XtsMover;
END_VAR
END_METHOD

METHOD DeregisterWithParent
VAR_INPUT
	Parent	: Core.I_ContainComponents;
END_VAR
END_METHOD

METHOD Disable
END_METHOD

METHOD Enable
END_METHOD

PROPERTY Enabled : BOOL
GET
END_GET
END_PROPERTY

METHOD GetMover : I_XtsMover
GetMover := NullObjects.XtsMover;
END_METHOD

METHOD IsMoverRegistered : BOOL
VAR_INPUT
	Mover : I_XtsMover;
END_VAR
END_METHOD

PROPERTY MoverIsPresent : BOOL
GET
END_GET
END_PROPERTY

PROPERTY MoverQueue : I_XtsMoverQueue
GET
END_GET
END_PROPERTY

PROPERTY Movers : I_XtsMoverEnumerator
GET
Movers := NullObjects.MoverCollection;
END_GET
SET
END_SET
END_PROPERTY

PROPERTY Name : Core.T_MaxString
GET
Name := 'Null  Xts Position Trigger';
END_GET
SET
END_SET
END_PROPERTY

PROPERTY Position : LREAL
GET
END_GET
SET
END_SET
END_PROPERTY

METHOD RegisterMover
VAR_INPUT
	Mover	: I_XtsMover;
END_VAR
END_METHOD

METHOD RegisterWithParent
VAR_INPUT
	Parent	: Core.I_ContainComponents;
END_VAR
END_METHOD

{attribute 'monitoring':='call'}
PROPERTY Status : I_XtsPositionTriggerStatus
GET
Status := NullObjects.XtsPositionTriggerStatus;
END_GET
END_PROPERTY

PROPERTY TracePublisher : I_XtsTracePublisher
GET
TracePublisher := NullObjects.MechatronicsTracePublisher;
END_GET
END_PROPERTY

END_FUNCTION_BLOCK

// _Internal/NullObjects/NullXtsPositionTriggerStatus
{attribute 'no_explicit_call' := 'This FB is a CLASS and must be accessed using methods or properties'}
{attribute 'conditionalshow'}
{warning disable C0094}
FUNCTION_BLOCK NullXtsPositionTriggerStatus IMPLEMENTS I_XtsPositionTriggerStatus, I_NullObject
VAR
END_VAR

{attribute 'monitoring':='call'}
//Number of Movers that have occurred and are in the current queue
PROPERTY NumberOfMoverEvents : UDINT
GET
END_GET
END_PROPERTY

{attribute 'monitoring' := 'call'}
(*Number of Movers Currently Registered to the Station*)
PROPERTY NumberOfMoversRegistered : UDINT
GET
END_GET
END_PROPERTY

END_FUNCTION_BLOCK

// _Internal/NullObjects/NullXtsStationStatus
{attribute 'no_explicit_call' := 'This FB is a CLASS and must be accessed using methods or properties'}
{attribute 'conditionalshow'}
{warning disable C0094}
FUNCTION_BLOCK NullXtsStationStatus IMPLEMENTS I_XtsStationStatus, I_NullObject
VAR
END_VAR

{attribute 'monitoring' := 'call'}
PROPERTY CurrentMoverId : UDINT
GET
END_GET
END_PROPERTY

{attribute 'monitoring' := 'call'}
PROPERTY CurrentMoverName : T_MaxString
GET
END_GET
END_PROPERTY

{attribute 'monitoring' := 'call'}
PROPERTY NumberOfMoversRegistered : UDINT
GET
END_GET
END_PROPERTY

END_FUNCTION_BLOCK

// _Internal/NullObjects/NullXtsSystem
{attribute 'no_explicit_call' := 'This FB is a CLASS and must be accessed using methods or properties'}
{attribute 'conditionalshow'}
{warning disable C0094}
{warning disable C0568}
FUNCTION_BLOCK NullXtsSystem IMPLEMENTS I_XtsSystem, I_NullObject
VAR
	_Config : NullXtsSystemConfiguration;
END_VAR

METHOD Accept
VAR_INPUT
	Visitor	: Core.I_ModuleVisitor;
END_VAR
END_METHOD

METHOD AcceptMoverVisitor
VAR_INPUT
	MoverVisitor	: I_XtsMoverVisitor;
END_VAR
END_METHOD

METHOD AcceptStationVisitor
VAR_INPUT
	StationVisitor : I_XtsStationVisitor;
END_VAR
END_METHOD

METHOD AcceptXtsModuleVisitor
VAR_INPUT
	XtsModuleVisitor : I_XtsModuleVisitor;
END_VAR
END_METHOD

METHOD AcceptXtsPartVisitor
VAR_INPUT
	XtsPartVisitor : I_XtsPartVisitor;
END_VAR
END_METHOD

METHOD AcceptXtsPositionTriggerVisitor
VAR_INPUT
	PositionTriggerVisitor : I_VisitXtsPositionTrigger;
END_VAR
END_METHOD

METHOD AcceptXtsZoneVisitor
VAR_INPUT
	ZoneVisitor : I_XtsZoneVisitor;
END_VAR
END_METHOD

PROPERTY AxesGroupRef : REFERENCE TO AXES_GROUP_REF
GET
END_GET
END_PROPERTY

{attribute 'monitoring' := 'call'}
PROPERTY Busy : BOOL
GET
END_GET
END_PROPERTY

{attribute 'monitoring' := 'call'}
PROPERTY CAGroupErrorId : UDINT
GET
END_GET
END_PROPERTY

{attribute 'monitoring' := 'call'}
PROPERTY CaGroupStatus : E_MoverGroupState
GET
END_GET
END_PROPERTY

{attribute 'monitoring' := 'call'}
PROPERTY CommandLog : I_XtsLocalLog
GET
CommandLog := NullObjects.MechatronicsLocalLog;
END_GET
END_PROPERTY

PROPERTY Components : Core.I_ComponentCollection
GET
END_GET
END_PROPERTY

{attribute 'monitoring' := 'call'}
PROPERTY Config : I_XtsSystemConfiguration
GET
Config := _Config;
END_GET
SET
END_SET
END_PROPERTY

PROPERTY CurrentTask : I_XtsTask
GET
CurrentTask := NullObjects.XtsTask;
END_GET
END_PROPERTY

METHOD CyclicLogic
END_METHOD

METHOD DeregisterComponent: RegistrationResult
VAR_INPUT
	Component	: Core.I_Component;
END_VAR
END_METHOD

METHOD DeregisterCyclic : RegistrationResult
VAR_INPUT
	Cyclic	: Core.I_Cyclic;
END_VAR
END_METHOD

METHOD DeregisterInitialize : RegistrationResult
VAR_INPUT
	Initializable	: Core.I_Initializable;
END_VAR
END_METHOD

METHOD DeregisterModule : RegistrationResult
VAR_INPUT
	Module	: Core.I_Module;
END_VAR
END_METHOD

METHOD DeregisterWithParent 
VAR_INPUT
	Parent	: Core.I_ContainModules;
END_VAR
END_METHOD

METHOD Disable
END_METHOD

METHOD DisableGroup
VAR_INPUT
END_VAR
END_METHOD

METHOD DisableMovers
VAR_INPUT
END_VAR
END_METHOD

METHOD Enable
END_METHOD

{attribute 'monitoring' := 'call'}
PROPERTY Enabled : BOOL
GET
END_GET
END_PROPERTY

METHOD EnableGroup
VAR_INPUT
END_VAR
END_METHOD

METHOD EnableMovers
VAR_INPUT
END_VAR
END_METHOD

PROPERTY Environment : I_TcIoXtsEnvironment
GET
END_GET
SET
END_SET
END_PROPERTY

{attribute 'monitoring' := 'call'}
PROPERTY Error : BOOL
GET
END_GET
END_PROPERTY

{attribute 'monitoring' := 'call'}
PROPERTY ErrorId : UDINT
GET
END_GET
END_PROPERTY

METHOD Initialize
END_METHOD

{attribute 'monitoring' := 'call'}
PROPERTY Initialized : BOOL
GET
END_GET
SET
END_SET
END_PROPERTY

{attribute 'monitoring' := 'call'}
PROPERTY ManualDiagnoser : REFERENCE TO ManualDebugger
GET
END_GET
END_PROPERTY

PROPERTY Modules : Core.I_ModuleCollection
GET
END_GET
END_PROPERTY

{attribute 'monitoring' := 'call'}
PROPERTY Movers : I_XtsMoverCollection
GET
Movers := NullObjects.MoverCollection;
END_GET
END_PROPERTY

{attribute 'monitoring' := 'call'}
PROPERTY MoversEnabled : BOOL
GET
END_GET
END_PROPERTY

{attribute 'monitoring' := 'call'}
PROPERTY Name : Core.T_MaxString
GET
END_GET
END_PROPERTY

{attribute 'monitoring' := 'call'}
PROPERTY Parameters : I_XtsParameterSet
GET
Parameters := NullObjects.XtsParameterSet;
END_GET
SET
END_SET
END_PROPERTY

PROPERTY Parts : I_XtsPartCollection
GET
Parts := NullObjects.XtsPartCollection;
END_GET
END_PROPERTY

PROPERTY PositionTriggers : I_XtsPositionTriggerCollection
GET
PositionTriggers := NullObjects.PositionTriggerCollection;
END_GET
END_PROPERTY

METHOD RegisterComponent : RegistrationResult
VAR_INPUT
	Component	: Core.I_Component;
END_VAR
END_METHOD

METHOD RegisterCyclic : RegistrationResult
VAR_INPUT
	Cyclic	: Core.I_Cyclic;
END_VAR
END_METHOD

METHOD RegisterInitialize : RegistrationResult
VAR_INPUT
	Initializable	: Core.I_Initializable;
END_VAR
END_METHOD

METHOD RegisterModule : RegistrationResult
VAR_INPUT
	Module	: Core.I_Module;
END_VAR
END_METHOD

METHOD RegisterWithParent 
VAR_INPUT
	Parent	: Core.I_ContainModules;
END_VAR
END_METHOD

METHOD Reset
END_METHOD

METHOD ResetCaGroup
VAR_INPUT
END_VAR
END_METHOD

METHOD ResetComponents : BOOL
END_METHOD

METHOD ResetModules : BOOL
END_METHOD

METHOD ResetMovers
VAR_INPUT
END_VAR
END_METHOD

METHOD RetriggerMoverDetection
END_METHOD

PROPERTY Stations : I_XtsStationCollection
GET
Stations := NullObjects.StationCollection;
END_GET
END_PROPERTY

{attribute 'monitoring' := 'call'}
PROPERTY Status : I_XtsSystemStatus
GET
Status := NullObjects.SystemStatus;
END_GET
END_PROPERTY

PROPERTY TracePublisher : I_XtsTracePublisher
GET
TracePublisher := NullObjects.MechatronicsTracePublisher;
END_GET
END_PROPERTY

PROPERTY Tracks : I_XtsTrackCollection
GET
Tracks := NullObjects.XtsTrackCollection;
END_GET
END_PROPERTY

METHOD TriggerMoverDetection
END_METHOD

METHOD TriggerMoverIdentification
END_METHOD

PROPERTY Utility : I_TcIoXtsProcessingUnit
GET
END_GET
SET
END_SET
END_PROPERTY

PROPERTY UtilityProperties : I_XtsSystemUtilityProperties
GET
END_GET
END_PROPERTY

{attribute 'monitoring' := 'call'}
PROPERTY XpuId : USINT
GET
END_GET
END_PROPERTY

PROPERTY XtsTasks : I_XtsTaskCollection
GET
XtsTasks := NullObjects.XtsSystemTasks;
END_GET
END_PROPERTY

PROPERTY Zones : I_XtsZoneCollection
GET
Zones := NullObjects.ZoneCollection;
END_GET
END_PROPERTY

END_FUNCTION_BLOCK

// _Internal/NullObjects/NullXtsSystemConfiguration
{attribute 'no_explicit_call' := 'This FB is a CLASS and must be accessed using methods or properties'}
{attribute 'conditionalshow'}
{warning disable C0094}
FUNCTION_BLOCK NullXtsSystemConfiguration IMPLEMENTS I_XtsSystemConfiguration, I_NullObject
VAR
END_VAR

{attribute 'monitoring' := 'call'}
PROPERTY CommandPositionTriggersOnDisable : BOOL
GET
END_GET
SET
END_SET
END_PROPERTY

{attribute 'monitoring' := 'call'}
PROPERTY CommandPositionTriggersOnEnable : BOOL
GET
END_GET
SET
END_SET
END_PROPERTY

{attribute 'monitoring' := 'call'}
PROPERTY CommandStationsOnDisable : BOOL
GET
END_GET
SET
END_SET
END_PROPERTY

{attribute 'monitoring' := 'call'}
PROPERTY CommandStationsOnEnable : BOOL
GET
END_GET
SET
END_SET
END_PROPERTY

END_FUNCTION_BLOCK

// _Internal/NullObjects/NullXtsSystemStatus
{attribute 'no_explicit_call' := 'This FB is a CLASS and must be accessed using methods or properties'}
{attribute 'conditionalshow'}
{warning disable C0094}
FUNCTION_BLOCK NullXtsSystemStatus IMPLEMENTS I_XtsSystemStatus,I_NullObject
VAR
END_VAR

METHOD CyclicLogic
END_METHOD

{attribute 'monitoring' := 'call'}
PROPERTY NumberOfMovers : UDINT
GET
END_GET
END_PROPERTY

{attribute 'monitoring' := 'call'}
PROPERTY NumberOfParts : UDINT
GET
END_GET
END_PROPERTY

{attribute 'monitoring' := 'call'}
PROPERTY NumberOfPositionTriggers : UDINT
GET
END_GET
END_PROPERTY

{attribute 'monitoring' := 'call'}
PROPERTY NumberOfStations : UDINT
GET
END_GET
END_PROPERTY

{attribute 'monitoring' := 'call'}
PROPERTY NumberOfTracks : UDINT
GET
END_GET
END_PROPERTY

{attribute 'monitoring' := 'call'}
PROPERTY NumberOfZones : UDINT
GET
END_GET
END_PROPERTY

{attribute 'monitoring' := 'call'}
PROPERTY NumberPartsNotReady : USINT
GET
END_GET
END_PROPERTY

{attribute 'monitoring' := 'call'}
PROPERTY NumberPartsReady : USINT
GET
END_GET
END_PROPERTY

{attribute 'monitoring' := 'call'}
PROPERTY Simulated : BOOL
GET
END_GET
END_PROPERTY

{attribute 'monitoring' := 'call'}
PROPERTY Vdc24Okay : BOOL
GET
END_GET
END_PROPERTY

{attribute 'monitoring' := 'call'}
PROPERTY Vdc48Okay : BOOL
GET
END_GET
END_PROPERTY

END_FUNCTION_BLOCK

